KUKA KRL program: unicorn_3.src

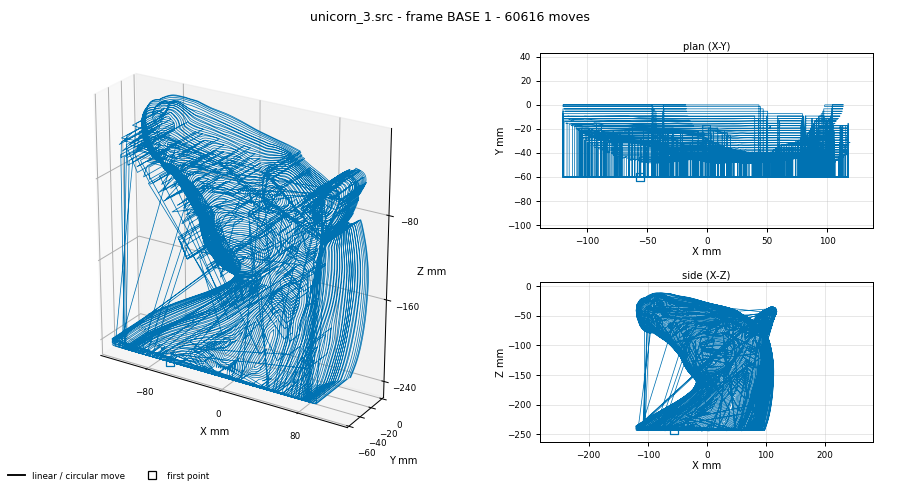
[picture p0: tool path of unicorn_3.src in frame BASE 1, 60616 of 60617 moves have a stored position in this frame; points joined in program order, loops and branches not executed]
&ACCESS RVP
&REL 1
&PARAM TEMPLATE = C:\KRC\Roboter\Template\vorgabe
&PARAM EDITMASK = *
DEF unicorn_3( )
EXT BAS (BAS_COMMAND :IN,REAL :IN )

INT INDX
FOR INDX=1 TO 6
	$ACC_AXIS[INDX]=50
	$VEL_AXIS[INDX]=20
ENDFOR

$VEL.ORI1=200
$VEL.ORI2=200
$ACC.ORI1=100
$ACC.ORI2=100

$VEL.CP = 0.2
$ACC.CP = 5

$IPO_MODE = #BASE
$APO.CDIS = 0.5
$ADVANCE = 5

$ACT_TOOL = 1
$TOOL=TOOL_DATA[1]
$ACT_BASE = 1
$BASE=BASE_DATA[1]

PTP {A1 30.0,A2 -100.0,A3 70.0,A4 0.0,A5 40.0,A6 0.0}

LIN {X -56.297,Y -60.000,Z -243.561,A -90.000,B 90.000,C 0.000} C_DIS
LIN {X -56.297,Y -47.308,Z -243.561,A -90.000,B 90.000,C 0.000} C_DIS
LIN {X -55.435,Y -47.308,Z -243.187,A -90.000,B 90.000,C 0.000} C_DIS
LIN {X -55.139,Y -47.308,Z -243.067,A -90.000,B 90.000,C 0.000} C_DIS
LIN {X -53.671,Y -47.308,Z -242.485,A -90.000,B 90.000,C 0.000} C_DIS
LIN {X -50.676,Y -47.308,Z -241.473,A -90.000,B 90.000,C 0.000} C_DIS
LIN {X -47.224,Y -47.308,Z -240.424,A -90.000,B 90.000,C 0.000} C_DIS
LIN {X -47.138,Y -47.308,Z -240.398,A -90.000,B 90.000,C 0.000} C_DIS
LIN {X -44.555,Y -47.308,Z -239.681,A -90.000,B 90.000,C 0.000} C_DIS
LIN {X -43.438,Y -47.308,Z -239.453,A -90.000,B 90.000,C 0.000} C_DIS
LIN {X -42.208,Y -47.308,Z -239.261,A -90.000,B 90.000,C 0.000} C_DIS
LIN {X -39.907,Y -47.308,Z -238.995,A -90.000,B 90.000,C 0.000} C_DIS
LIN {X -38.204,Y -47.308,Z -238.801,A -90.000,B 90.000,C 0.000} C_DIS
LIN {X -37.466,Y -47.308,Z -238.748,A -90.000,B 90.000,C 0.000} C_DIS
LIN {X -37.229,Y -47.308,Z -238.745,A -90.000,B 90.000,C 0.000} C_DIS
LIN {X -34.457,Y -47.308,Z -239.098,A -90.000,B 90.000,C 0.000} C_DIS
LIN {X -34.198,Y -47.308,Z -239.146,A -90.000,B 90.000,C 0.000} C_DIS
LIN {X -32.605,Y -47.308,Z -239.457,A -90.000,B 90.000,C 0.000} C_DIS
LIN {X -32.434,Y -47.308,Z -239.513,A -90.000,B 90.000,C 0.000} C_DIS
LIN {X -31.010,Y -47.308,Z -240.218,A -90.000,B 90.000,C 0.000} C_DIS
LIN {X -29.625,Y -47.308,Z -241.071,A -90.000,B 90.000,C 0.000} C_DIS
LIN {X -29.477,Y -47.308,Z -241.172,A -90.000,B 90.000,C 0.000} C_DIS
LIN {X -28.409,Y -47.308,Z -242.294,A -90.000,B 90.000,C 0.000} C_DIS
LIN {X -28.294,Y -47.308,Z -242.432,A -90.000,B 90.000,C 0.000} C_DIS
LIN {X -27.412,Y -47.308,Z -243.561,A -90.000,B 90.000,C 0.000} C_DIS
LIN {X -27.429,Y -47.311,Z -243.561,A -90.000,B 90.000,C 0.000} C_DIS
LIN {X -29.070,Y -47.511,Z -243.561,A -90.000,B 90.000,C 0.000} C_DIS
LIN {X -32.555,Y -47.888,Z -243.561,A -90.000,B 90.000,C 0.000} C_DIS
LIN {X -32.864,Y -47.915,Z -243.561,A -90.000,B 90.000,C 0.000} C_DIS
LIN {X -36.464,Y -48.174,Z -243.561,A -90.000,B 90.000,C 0.000} C_DIS
LIN {X -38.036,Y -48.261,Z -243.561,A -90.000,B 90.000,C 0.000} C_DIS
LIN {X -38.687,Y -48.281,Z -243.561,A -90.000,B 90.000,C 0.000} C_DIS
LIN {X -40.659,Y -48.330,Z -243.561,A -90.000,B 90.000,C 0.000} C_DIS
LIN {X -43.801,Y -48.366,Z -243.561,A -90.000,B 90.000,C 0.000} C_DIS
LIN {X -43.989,Y -48.366,Z -243.561,A -90.000,B 90.000,C 0.000} C_DIS
LIN {X -44.713,Y -48.344,Z -243.561,A -90.000,B 90.000,C 0.000} C_DIS
LIN {X -46.996,Y -48.250,Z -243.561,A -90.000,B 90.000,C 0.000} C_DIS
LIN {X -49.101,Y -48.148,Z -243.561,A -90.000,B 90.000,C 0.000} C_DIS
LIN {X -49.262,Y -48.138,Z -243.561,A -90.000,B 90.000,C 0.000} C_DIS
LIN {X -49.887,Y -48.091,Z -243.561,A -90.000,B 90.000,C 0.000} C_DIS
LIN {X -50.048,Y -48.076,Z -243.561,A -90.000,B 90.000,C 0.000} C_DIS
LIN {X -51.629,Y -47.893,Z -243.561,A -90.000,B 90.000,C 0.000} C_DIS
LIN {X -55.147,Y -47.500,Z -243.561,A -90.000,B 90.000,C 0.000} C_DIS
LIN {X -55.949,Y -47.375,Z -243.561,A -90.000,B 90.000,C 0.000} C_DIS
LIN {X -56.297,Y -47.308,Z -243.561,A -90.000,B 90.000,C 0.000} C_DIS
LIN {X -56.297,Y -60.000,Z -243.561,A -90.000,B 90.000,C 0.000} C_DIS
LIN {X -44.362,Y -60.000,Z -241.627,A -90.000,B 90.000,C 0.000} C_DIS
LIN {X -44.362,Y -47.846,Z -241.627,A -90.000,B 90.000,C 0.000} C_DIS
LIN {X -44.089,Y -47.838,Z -241.555,A -90.000,B 90.000,C 0.000} C_DIS
LIN {X -43.472,Y -47.831,Z -241.430,A -90.000,B 90.000,C 0.000} C_DIS
LIN {X -43.074,Y -47.823,Z -241.352,A -90.000,B 90.000,C 0.000} C_DIS
LIN {X -41.969,Y -47.812,Z -241.182,A -90.000,B 90.000,C 0.000} C_DIS
LIN {X -40.544,Y -47.812,Z -241.017,A -90.000,B 90.000,C 0.000} C_DIS
LIN {X -40.270,Y -47.806,Z -240.987,A -90.000,B 90.000,C 0.000} C_DIS
LIN {X -39.113,Y -47.767,Z -240.864,A -90.000,B 90.000,C 0.000} C_DIS
LIN {X -38.023,Y -47.717,Z -240.751,A -90.000,B 90.000,C 0.000} C_DIS
LIN {X -37.379,Y -47.693,Z -240.710,A -90.000,B 90.000,C 0.000} C_DIS
LIN {X -37.343,Y -47.692,Z -240.710,A -90.000,B 90.000,C 0.000} C_DIS
LIN {X -35.486,Y -47.692,Z -240.946,A -90.000,B 90.000,C 0.000} C_DIS
LIN {X -34.760,Y -47.683,Z -241.040,A -90.000,B 90.000,C 0.000} C_DIS
LIN {X -34.515,Y -47.679,Z -241.086,A -90.000,B 90.000,C 0.000} C_DIS
LIN {X -33.149,Y -47.622,Z -241.363,A -90.000,B 90.000,C 0.000} C_DIS
LIN {X -32.709,Y -47.622,Z -241.581,A -90.000,B 90.000,C 0.000} C_DIS
LIN {X -35.186,Y -47.796,Z -241.582,A -90.000,B 90.000,C 0.000} C_DIS
LIN {X -35.416,Y -47.809,Z -241.582,A -90.000,B 90.000,C 0.000} C_DIS
LIN {X -35.606,Y -47.816,Z -241.583,A -90.000,B 90.000,C 0.000} C_DIS
LIN {X -35.738,Y -47.821,Z -241.584,A -90.000,B 90.000,C 0.000} C_DIS
LIN {X -36.488,Y -47.842,Z -241.589,A -90.000,B 90.000,C 0.000} C_DIS
LIN {X -38.216,Y -47.887,Z -241.598,A -90.000,B 90.000,C 0.000} C_DIS
LIN {X -39.566,Y -47.921,Z -241.598,A -90.000,B 90.000,C 0.000} C_DIS
LIN {X -41.163,Y -47.939,Z -241.601,A -90.000,B 90.000,C 0.000} C_DIS
LIN {X -41.336,Y -47.939,Z -241.602,A -90.000,B 90.000,C 0.000} C_DIS
LIN {X -43.583,Y -47.877,Z -241.622,A -90.000,B 90.000,C 0.000} C_DIS
LIN {X -44.113,Y -47.856,Z -241.626,A -90.000,B 90.000,C 0.000} C_DIS
LIN {X -44.362,Y -47.846,Z -241.627,A -90.000,B 90.000,C 0.000} C_DIS
LIN {X -44.362,Y -60.000,Z -241.627,A -90.000,B 90.000,C 0.000} C_DIS
LIN {X 92.568,Y -60.000,Z -59.359,A -90.000,B 90.000,C 0.000} C_DIS
LIN {X 92.568,Y -51.610,Z -59.359,A -90.000,B 90.000,C 0.000} C_DIS
LIN {X 92.745,Y -51.646,Z -59.003,A -90.000,B 90.000,C 0.000} C_DIS
LIN {X 92.870,Y -51.669,Z -58.752,A -90.000,B 90.000,C 0.000} C_DIS
LIN {X 92.953,Y -51.684,Z -58.585,A -90.000,B 90.000,C 0.000} C_DIS
LIN {X 92.974,Y -51.688,Z -58.543,A -90.000,B 90.000,C 0.000} C_DIS
LIN {X 93.175,Y -51.715,Z -58.224,A -90.000,B 90.000,C 0.000} C_DIS
LIN {X 93.326,Y -51.727,Z -57.987,A -90.000,B 90.000,C 0.000} C_DIS
LIN {X 93.444,Y -51.726,Z -57.807,A -90.000,B 90.000,C 0.000} C_DIS
LIN {X 93.456,Y -51.725,Z -57.788,A -90.000,B 90.000,C 0.000} C_DIS
LIN {X 93.639,Y -51.720,Z -57.654,A -90.000,B 90.000,C 0.000} C_DIS
LIN {X 95.632,Y -51.629,Z -56.194,A -90.000,B 90.000,C 0.000} C_DIS
LIN {X 95.618,Y -51.636,Z -56.312,A -90.000,B 90.000,C 0.000} C_DIS
LIN {X 95.580,Y -51.642,Z -56.475,A -90.000,B 90.000,C 0.000} C_DIS
LIN {X 95.278,Y -51.660,Z -56.893,A -90.000,B 90.000,C 0.000} C_DIS
LIN {X 94.891,Y -51.678,Z -57.426,A -90.000,B 90.000,C 0.000} C_DIS
LIN {X 94.530,Y -51.696,Z -57.901,A -90.000,B 90.000,C 0.000} C_DIS
LIN {X 94.459,Y -51.699,Z -58.007,A -90.000,B 90.000,C 0.000} C_DIS
LIN {X 94.229,Y -51.708,Z -58.379,A -90.000,B 90.000,C 0.000} C_DIS
LIN {X 94.134,Y -51.708,Z -58.531,A -90.000,B 90.000,C 0.000} C_DIS
LIN {X 93.995,Y -51.711,Z -58.607,A -90.000,B 90.000,C 0.000} C_DIS
LIN {X 93.858,Y -51.710,Z -58.680,A -90.000,B 90.000,C 0.000} C_DIS
LIN {X 93.698,Y -51.705,Z -58.766,A -90.000,B 90.000,C 0.000} C_DIS
LIN {X 93.242,Y -51.670,Z -59.005,A -90.000,B 90.000,C 0.000} C_DIS
LIN {X 92.568,Y -51.610,Z -59.359,A -90.000,B 90.000,C 0.000} C_DIS
LIN {X 92.601,Y -51.623,Z -59.288,A -90.000,B 90.000,C 0.000} C_DIS
LIN {X 92.662,Y -51.637,Z -59.142,A -90.000,B 90.000,C 0.000} C_DIS
LIN {X 92.713,Y -51.650,Z -58.992,A -90.000,B 90.000,C 0.000} C_DIS
LIN {X 92.755,Y -51.661,Z -58.836,A -90.000,B 90.000,C 0.000} C_DIS
LIN {X 92.773,Y -51.666,Z -58.757,A -90.000,B 90.000,C 0.000} C_DIS
LIN {X 92.804,Y -51.673,Z -58.596,A -90.000,B 90.000,C 0.000} C_DIS
LIN {X 92.830,Y -51.679,Z -58.432,A -90.000,B 90.000,C 0.000} C_DIS
LIN {X 92.861,Y -51.683,Z -58.271,A -90.000,B 90.000,C 0.000} C_DIS
LIN {X 92.886,Y -51.683,Z -58.108,A -90.000,B 90.000,C 0.000} C_DIS
LIN {X 92.916,Y -51.679,Z -57.858,A -90.000,B 90.000,C 0.000} C_DIS
LIN {X 92.945,Y -51.662,Z -57.519,A -90.000,B 90.000,C 0.000} C_DIS
LIN {X 92.964,Y -51.658,Z -57.446,A -90.000,B 90.000,C 0.000} C_DIS
LIN {X 93.093,Y -51.597,Z -56.846,A -90.000,B 90.000,C 0.000} C_DIS
LIN {X 93.110,Y -51.588,Z -56.773,A -90.000,B 90.000,C 0.000} C_DIS
LIN {X 93.210,Y -51.543,Z -56.418,A -90.000,B 90.000,C 0.000} C_DIS
LIN {X 93.299,Y -51.507,Z -56.138,A -90.000,B 90.000,C 0.000} C_DIS
LIN {X 93.374,Y -51.480,Z -55.933,A -90.000,B 90.000,C 0.000} C_DIS
LIN {X 93.459,Y -51.453,Z -55.733,A -90.000,B 90.000,C 0.000} C_DIS
LIN {X 93.556,Y -51.427,Z -55.540,A -90.000,B 90.000,C 0.000} C_DIS
LIN {X 93.629,Y -51.409,Z -55.416,A -90.000,B 90.000,C 0.000} C_DIS
LIN {X 93.668,Y -51.400,Z -55.356,A -90.000,B 90.000,C 0.000} C_DIS
LIN {X 93.752,Y -51.382,Z -55.238,A -90.000,B 90.000,C 0.000} C_DIS
LIN {X 93.797,Y -51.373,Z -55.180,A -90.000,B 90.000,C 0.000} C_DIS
LIN {X 93.891,Y -51.356,Z -55.073,A -90.000,B 90.000,C 0.000} C_DIS
LIN {X 93.998,Y -51.337,Z -54.967,A -90.000,B 90.000,C 0.000} C_DIS
LIN {X 94.055,Y -51.328,Z -54.915,A -90.000,B 90.000,C 0.000} C_DIS
LIN {X 94.178,Y -51.308,Z -54.816,A -90.000,B 90.000,C 0.000} C_DIS
LIN {X 94.616,Y -51.308,Z -54.490,A -90.000,B 90.000,C 0.000} C_DIS
LIN {X 94.876,Y -51.308,Z -54.360,A -90.000,B 90.000,C 0.000} C_DIS
LIN {X 95.150,Y -51.308,Z -54.278,A -90.000,B 90.000,C 0.000} C_DIS
LIN {X 96.092,Y -51.308,Z -54.069,A -90.000,B 90.000,C 0.000} C_DIS
LIN {X 96.329,Y -51.308,Z -54.067,A -90.000,B 90.000,C 0.000} C_DIS
LIN {X 96.828,Y -51.308,Z -54.127,A -90.000,B 90.000,C 0.000} C_DIS
LIN {X 96.999,Y -51.308,Z -54.183,A -90.000,B 90.000,C 0.000} C_DIS
LIN {X 97.188,Y -51.308,Z -54.264,A -90.000,B 90.000,C 0.000} C_DIS
LIN {X 97.336,Y -51.308,Z -54.364,A -90.000,B 90.000,C 0.000} C_DIS
LIN {X 97.572,Y -51.308,Z -54.640,A -90.000,B 90.000,C 0.000} C_DIS
LIN {X 97.647,Y -51.308,Z -54.730,A -90.000,B 90.000,C 0.000} C_DIS
LIN {X 97.720,Y -51.308,Z -54.894,A -90.000,B 90.000,C 0.000} C_DIS
LIN {X 97.745,Y -51.308,Z -55.071,A -90.000,B 90.000,C 0.000} C_DIS
LIN {X 97.779,Y -51.308,Z -55.468,A -90.000,B 90.000,C 0.000} C_DIS
LIN {X 97.763,Y -51.308,Z -55.657,A -90.000,B 90.000,C 0.000} C_DIS
LIN {X 97.699,Y -51.308,Z -55.885,A -90.000,B 90.000,C 0.000} C_DIS
LIN {X 97.636,Y -51.308,Z -56.084,A -90.000,B 90.000,C 0.000} C_DIS
LIN {X 97.562,Y -51.308,Z -56.670,A -90.000,B 90.000,C 0.000} C_DIS
LIN {X 97.474,Y -51.308,Z -57.034,A -90.000,B 90.000,C 0.000} C_DIS
LIN {X 97.439,Y -51.308,Z -57.158,A -90.000,B 90.000,C 0.000} C_DIS
LIN {X 97.395,Y -51.308,Z -57.279,A -90.000,B 90.000,C 0.000} C_DIS
LIN {X 97.335,Y -51.308,Z -57.393,A -90.000,B 90.000,C 0.000} C_DIS
LIN {X 97.271,Y -51.308,Z -57.504,A -90.000,B 90.000,C 0.000} C_DIS
LIN {X 96.478,Y -51.308,Z -58.586,A -90.000,B 90.000,C 0.000} C_DIS
LIN {X 96.123,Y -51.308,Z -59.047,A -90.000,B 90.000,C 0.000} C_DIS
LIN {X 95.658,Y -51.308,Z -59.790,A -90.000,B 90.000,C 0.000} C_DIS
LIN {X 95.506,Y -51.308,Z -59.971,A -90.000,B 90.000,C 0.000} C_DIS
LIN {X 95.321,Y -51.308,Z -60.117,A -90.000,B 90.000,C 0.000} C_DIS
LIN {X 92.838,Y -51.308,Z -61.461,A -90.000,B 90.000,C 0.000} C_DIS
LIN {X 92.625,Y -51.308,Z -61.565,A -90.000,B 90.000,C 0.000} C_DIS
LIN {X 92.395,Y -51.308,Z -61.622,A -90.000,B 90.000,C 0.000} C_DIS
LIN {X 92.140,Y -51.308,Z -61.630,A -90.000,B 90.000,C 0.000} C_DIS
LIN {X 91.914,Y -51.308,Z -61.589,A -90.000,B 90.000,C 0.000} C_DIS
LIN {X 91.898,Y -51.308,Z -61.586,A -90.000,B 90.000,C 0.000} C_DIS
LIN {X 91.679,Y -51.308,Z -61.496,A -90.000,B 90.000,C 0.000} C_DIS
LIN {X 91.018,Y -51.308,Z -61.119,A -90.000,B 90.000,C 0.000} C_DIS
LIN {X 90.824,Y -51.308,Z -60.986,A -90.000,B 90.000,C 0.000} C_DIS
LIN {X 90.661,Y -51.308,Z -60.814,A -90.000,B 90.000,C 0.000} C_DIS
LIN {X 90.538,Y -51.308,Z -60.612,A -90.000,B 90.000,C 0.000} C_DIS
LIN {X 90.499,Y -51.308,Z -60.517,A -90.000,B 90.000,C 0.000} C_DIS
LIN {X 90.453,Y -51.308,Z -60.387,A -90.000,B 90.000,C 0.000} C_DIS
LIN {X 90.417,Y -51.308,Z -60.274,A -90.000,B 90.000,C 0.000} C_DIS
LIN {X 90.383,Y -51.308,Z -60.021,A -90.000,B 90.000,C 0.000} C_DIS
LIN {X 90.375,Y -51.308,Z -59.750,A -90.000,B 90.000,C 0.000} C_DIS
LIN {X 90.395,Y -51.308,Z -59.514,A -90.000,B 90.000,C 0.000} C_DIS
LIN {X 90.464,Y -51.308,Z -59.287,A -90.000,B 90.000,C 0.000} C_DIS
LIN {X 90.637,Y -51.308,Z -58.788,A -90.000,B 90.000,C 0.000} C_DIS
LIN {X 91.272,Y -51.308,Z -57.559,A -90.000,B 90.000,C 0.000} C_DIS
LIN {X 91.425,Y -51.308,Z -57.322,A -90.000,B 90.000,C 0.000} C_DIS
LIN {X 91.901,Y -51.308,Z -56.593,A -90.000,B 90.000,C 0.000} C_DIS
LIN {X 92.004,Y -51.308,Z -56.475,A -90.000,B 90.000,C 0.000} C_DIS
LIN {X 92.101,Y -51.308,Z -56.370,A -90.000,B 90.000,C 0.000} C_DIS
LIN {X 92.222,Y -51.308,Z -56.269,A -90.000,B 90.000,C 0.000} C_DIS
LIN {X 94.178,Y -51.308,Z -54.816,A -90.000,B 90.000,C 0.000} C_DIS
LIN {X 94.209,Y -51.312,Z -54.791,A -90.000,B 90.000,C 0.000} C_DIS
LIN {X 94.266,Y -51.308,Z -54.736,A -90.000,B 90.000,C 0.000} C_DIS
LIN {X 94.318,Y -51.301,Z -54.674,A -90.000,B 90.000,C 0.000} C_DIS
LIN {X 94.365,Y -51.290,Z -54.604,A -90.000,B 90.000,C 0.000} C_DIS
LIN {X 94.407,Y -51.276,Z -54.529,A -90.000,B 90.000,C 0.000} C_DIS
LIN {X 94.444,Y -51.260,Z -54.447,A -90.000,B 90.000,C 0.000} C_DIS
LIN {X 94.528,Y -51.204,Z -54.231,A -90.000,B 90.000,C 0.000} C_DIS
LIN {X 94.560,Y -51.177,Z -54.143,A -90.000,B 90.000,C 0.000} C_DIS
LIN {X 94.644,Y -51.086,Z -53.871,A -90.000,B 90.000,C 0.000} C_DIS
LIN {X 94.670,Y -51.055,Z -53.778,A -90.000,B 90.000,C 0.000} C_DIS
LIN {X 94.787,Y -50.899,Z -53.300,A -90.000,B 90.000,C 0.000} C_DIS
LIN {X 94.864,Y -50.807,Z -53.022,A -90.000,B 90.000,C 0.000} C_DIS
LIN {X 94.924,Y -50.748,Z -52.847,A -90.000,B 90.000,C 0.000} C_DIS
LIN {X 94.976,Y -50.707,Z -52.729,A -90.000,B 90.000,C 0.000} C_DIS
LIN {X 95.016,Y -50.681,Z -52.656,A -90.000,B 90.000,C 0.000} C_DIS
LIN {X 95.058,Y -50.656,Z -52.589,A -90.000,B 90.000,C 0.000} C_DIS
LIN {X 95.106,Y -50.631,Z -52.528,A -90.000,B 90.000,C 0.000} C_DIS
LIN {X 95.157,Y -50.607,Z -52.473,A -90.000,B 90.000,C 0.000} C_DIS
LIN {X 95.214,Y -50.584,Z -52.425,A -90.000,B 90.000,C 0.000} C_DIS
LIN {X 95.277,Y -50.560,Z -52.385,A -90.000,B 90.000,C 0.000} C_DIS
LIN {X 95.346,Y -50.536,Z -52.354,A -90.000,B 90.000,C 0.000} C_DIS
LIN {X 95.383,Y -50.524,Z -52.342,A -90.000,B 90.000,C 0.000} C_DIS
LIN {X 95.398,Y -50.526,Z -52.338,A -90.000,B 90.000,C 0.000} C_DIS
LIN {X 95.699,Y -50.560,Z -52.257,A -90.000,B 90.000,C 0.000} C_DIS
LIN {X 95.879,Y -50.584,Z -52.217,A -90.000,B 90.000,C 0.000} C_DIS
LIN {X 96.072,Y -50.619,Z -52.192,A -90.000,B 90.000,C 0.000} C_DIS
LIN {X 96.251,Y -50.654,Z -52.178,A -90.000,B 90.000,C 0.000} C_DIS
LIN {X 96.315,Y -50.664,Z -52.174,A -90.000,B 90.000,C 0.000} C_DIS
LIN {X 96.555,Y -50.706,Z -52.173,A -90.000,B 90.000,C 0.000} C_DIS
LIN {X 96.842,Y -50.762,Z -52.191,A -90.000,B 90.000,C 0.000} C_DIS
LIN {X 96.936,Y -50.779,Z -52.197,A -90.000,B 90.000,C 0.000} C_DIS
LIN {X 97.072,Y -50.798,Z -52.208,A -90.000,B 90.000,C 0.000} C_DIS
LIN {X 97.235,Y -50.822,Z -52.230,A -90.000,B 90.000,C 0.000} C_DIS
LIN {X 97.288,Y -50.829,Z -52.240,A -90.000,B 90.000,C 0.000} C_DIS
LIN {X 97.451,Y -50.854,Z -52.281,A -90.000,B 90.000,C 0.000} C_DIS
LIN {X 97.636,Y -50.884,Z -52.335,A -90.000,B 90.000,C 0.000} C_DIS
LIN {X 97.768,Y -50.897,Z -52.383,A -90.000,B 90.000,C 0.000} C_DIS
LIN {X 97.864,Y -50.907,Z -52.422,A -90.000,B 90.000,C 0.000} C_DIS
LIN {X 97.959,Y -50.913,Z -52.461,A -90.000,B 90.000,C 0.000} C_DIS
LIN {X 98.051,Y -50.919,Z -52.502,A -90.000,B 90.000,C 0.000} C_DIS
LIN {X 98.097,Y -50.923,Z -52.524,A -90.000,B 90.000,C 0.000} C_DIS
LIN {X 98.193,Y -50.933,Z -52.576,A -90.000,B 90.000,C 0.000} C_DIS
LIN {X 98.271,Y -50.942,Z -52.623,A -90.000,B 90.000,C 0.000} C_DIS
LIN {X 98.456,Y -50.952,Z -52.746,A -90.000,B 90.000,C 0.000} C_DIS
LIN {X 98.501,Y -50.952,Z -52.778,A -90.000,B 90.000,C 0.000} C_DIS
LIN {X 98.610,Y -50.953,Z -52.864,A -90.000,B 90.000,C 0.000} C_DIS
LIN {X 98.641,Y -50.954,Z -52.891,A -90.000,B 90.000,C 0.000} C_DIS
LIN {X 98.705,Y -50.952,Z -52.950,A -90.000,B 90.000,C 0.000} C_DIS
LIN {X 98.809,Y -50.952,Z -53.059,A -90.000,B 90.000,C 0.000} C_DIS
LIN {X 99.055,Y -50.948,Z -53.347,A -90.000,B 90.000,C 0.000} C_DIS
LIN {X 99.196,Y -50.939,Z -53.520,A -90.000,B 90.000,C 0.000} C_DIS
LIN {X 99.250,Y -50.934,Z -53.594,A -90.000,B 90.000,C 0.000} C_DIS
LIN {X 99.296,Y -50.928,Z -53.664,A -90.000,B 90.000,C 0.000} C_DIS
LIN {X 99.365,Y -50.920,Z -53.781,A -90.000,B 90.000,C 0.000} C_DIS
LIN {X 99.410,Y -50.911,Z -53.872,A -90.000,B 90.000,C 0.000} C_DIS
LIN {X 99.508,Y -50.891,Z -54.101,A -90.000,B 90.000,C 0.000} C_DIS
LIN {X 99.574,Y -50.876,Z -54.280,A -90.000,B 90.000,C 0.000} C_DIS
LIN {X 99.601,Y -50.865,Z -54.378,A -90.000,B 90.000,C 0.000} C_DIS
LIN {X 99.621,Y -50.850,Z -54.474,A -90.000,B 90.000,C 0.000} C_DIS
LIN {X 99.639,Y -50.841,Z -54.578,A -90.000,B 90.000,C 0.000} C_DIS
LIN {X 99.671,Y -50.821,Z -54.837,A -90.000,B 90.000,C 0.000} C_DIS
LIN {X 99.683,Y -50.811,Z -54.996,A -90.000,B 90.000,C 0.000} C_DIS
LIN {X 99.703,Y -50.785,Z -55.307,A -90.000,B 90.000,C 0.000} C_DIS
LIN {X 99.697,Y -50.751,Z -55.568,A -90.000,B 90.000,C 0.000} C_DIS
LIN {X 99.668,Y -50.720,Z -55.818,A -90.000,B 90.000,C 0.000} C_DIS
LIN {X 99.647,Y -50.705,Z -55.953,A -90.000,B 90.000,C 0.000} C_DIS
LIN {X 99.614,Y -50.692,Z -56.100,A -90.000,B 90.000,C 0.000} C_DIS
LIN {X 99.527,Y -50.673,Z -56.389,A -90.000,B 90.000,C 0.000} C_DIS
LIN {X 99.494,Y -50.667,Z -56.491,A -90.000,B 90.000,C 0.000} C_DIS
LIN {X 99.480,Y -50.658,Z -56.578,A -90.000,B 90.000,C 0.000} C_DIS
LIN {X 99.413,Y -50.624,Z -56.993,A -90.000,B 90.000,C 0.000} C_DIS
LIN {X 99.380,Y -50.616,Z -57.135,A -90.000,B 90.000,C 0.000} C_DIS
LIN {X 99.310,Y -50.598,Z -57.393,A -90.000,B 90.000,C 0.000} C_DIS
LIN {X 99.255,Y -50.580,Z -57.579,A -90.000,B 90.000,C 0.000} C_DIS
LIN {X 99.220,Y -50.571,Z -57.689,A -90.000,B 90.000,C 0.000} C_DIS
LIN {X 99.158,Y -50.567,Z -57.865,A -90.000,B 90.000,C 0.000} C_DIS
LIN {X 99.137,Y -50.567,Z -57.923,A -90.000,B 90.000,C 0.000} C_DIS
LIN {X 99.056,Y -50.570,Z -58.113,A -90.000,B 90.000,C 0.000} C_DIS
LIN {X 98.948,Y -50.580,Z -58.324,A -90.000,B 90.000,C 0.000} C_DIS
LIN {X 98.834,Y -50.590,Z -58.524,A -90.000,B 90.000,C 0.000} C_DIS
LIN {X 98.810,Y -50.593,Z -58.562,A -90.000,B 90.000,C 0.000} C_DIS
LIN {X 98.626,Y -50.600,Z -58.820,A -90.000,B 90.000,C 0.000} C_DIS
LIN {X 98.455,Y -50.599,Z -59.052,A -90.000,B 90.000,C 0.000} C_DIS
LIN {X 97.963,Y -50.613,Z -59.733,A -90.000,B 90.000,C 0.000} C_DIS
LIN {X 97.668,Y -50.626,Z -60.122,A -90.000,B 90.000,C 0.000} C_DIS
LIN {X 97.412,Y -50.622,Z -60.527,A -90.000,B 90.000,C 0.000} C_DIS
LIN {X 97.250,Y -50.616,Z -60.784,A -90.000,B 90.000,C 0.000} C_DIS
LIN {X 97.107,Y -50.621,Z -60.985,A -90.000,B 90.000,C 0.000} C_DIS
LIN {X 97.084,Y -50.622,Z -61.013,A -90.000,B 90.000,C 0.000} C_DIS
LIN {X 96.902,Y -50.619,Z -61.228,A -90.000,B 90.000,C 0.000} C_DIS
LIN {X 96.862,Y -50.619,Z -61.270,A -90.000,B 90.000,C 0.000} C_DIS
LIN {X 96.805,Y -50.616,Z -61.326,A -90.000,B 90.000,C 0.000} C_DIS
LIN {X 96.663,Y -50.615,Z -61.448,A -90.000,B 90.000,C 0.000} C_DIS
LIN {X 96.417,Y -50.620,Z -61.641,A -90.000,B 90.000,C 0.000} C_DIS
LIN {X 96.326,Y -50.624,Z -61.705,A -90.000,B 90.000,C 0.000} C_DIS
LIN {X 96.217,Y -50.632,Z -61.772,A -90.000,B 90.000,C 0.000} C_DIS
LIN {X 94.915,Y -50.736,Z -62.516,A -90.000,B 90.000,C 0.000} C_DIS
LIN {X 94.357,Y -50.764,Z -62.827,A -90.000,B 90.000,C 0.000} C_DIS
LIN {X 94.108,Y -50.765,Z -62.962,A -90.000,B 90.000,C 0.000} C_DIS
LIN {X 93.876,Y -50.752,Z -63.083,A -90.000,B 90.000,C 0.000} C_DIS
LIN {X 93.676,Y -50.727,Z -63.181,A -90.000,B 90.000,C 0.000} C_DIS
LIN {X 93.468,Y -50.706,Z -63.275,A -90.000,B 90.000,C 0.000} C_DIS
LIN {X 93.374,Y -50.697,Z -63.315,A -90.000,B 90.000,C 0.000} C_DIS
LIN {X 93.320,Y -50.692,Z -63.336,A -90.000,B 90.000,C 0.000} C_DIS
LIN {X 93.081,Y -50.681,Z -63.408,A -90.000,B 90.000,C 0.000} C_DIS
LIN {X 92.834,Y -50.676,Z -63.467,A -90.000,B 90.000,C 0.000} C_DIS
LIN {X 92.710,Y -50.675,Z -63.492,A -90.000,B 90.000,C 0.000} C_DIS
LIN {X 92.439,Y -50.684,Z -63.521,A -90.000,B 90.000,C 0.000} C_DIS
LIN {X 92.191,Y -50.695,Z -63.533,A -90.000,B 90.000,C 0.000} C_DIS
LIN {X 92.043,Y -50.695,Z -63.531,A -90.000,B 90.000,C 0.000} C_DIS
LIN {X 91.915,Y -50.697,Z -63.521,A -90.000,B 90.000,C 0.000} C_DIS
LIN {X 91.790,Y -50.698,Z -63.502,A -90.000,B 90.000,C 0.000} C_DIS
LIN {X 91.504,Y -50.701,Z -63.450,A -90.000,B 90.000,C 0.000} C_DIS
LIN {X 91.501,Y -50.701,Z -63.450,A -90.000,B 90.000,C 0.000} C_DIS
LIN {X 91.290,Y -50.709,Z -63.394,A -90.000,B 90.000,C 0.000} C_DIS
LIN {X 91.171,Y -50.721,Z -63.354,A -90.000,B 90.000,C 0.000} C_DIS
LIN {X 90.938,Y -50.748,Z -63.267,A -90.000,B 90.000,C 0.000} C_DIS
LIN {X 90.853,Y -50.753,Z -63.231,A -90.000,B 90.000,C 0.000} C_DIS
LIN {X 90.710,Y -50.766,Z -63.160,A -90.000,B 90.000,C 0.000} C_DIS
LIN {X 90.514,Y -50.783,Z -63.053,A -90.000,B 90.000,C 0.000} C_DIS
LIN {X 90.315,Y -50.791,Z -62.942,A -90.000,B 90.000,C 0.000} C_DIS
LIN {X 90.061,Y -50.784,Z -62.795,A -90.000,B 90.000,C 0.000} C_DIS
LIN {X 89.938,Y -50.780,Z -62.717,A -90.000,B 90.000,C 0.000} C_DIS
LIN {X 89.675,Y -50.776,Z -62.534,A -90.000,B 90.000,C 0.000} C_DIS
LIN {X 89.573,Y -50.779,Z -62.454,A -90.000,B 90.000,C 0.000} C_DIS
LIN {X 89.481,Y -50.783,Z -62.371,A -90.000,B 90.000,C 0.000} C_DIS
LIN {X 89.316,Y -50.783,Z -62.200,A -90.000,B 90.000,C 0.000} C_DIS
LIN {X 89.203,Y -50.774,Z -62.074,A -90.000,B 90.000,C 0.000} C_DIS
LIN {X 89.142,Y -50.769,Z -61.997,A -90.000,B 90.000,C 0.000} C_DIS
LIN {X 89.101,Y -50.764,Z -61.941,A -90.000,B 90.000,C 0.000} C_DIS
LIN {X 89.021,Y -50.755,Z -61.816,A -90.000,B 90.000,C 0.000} C_DIS
LIN {X 88.901,Y -50.739,Z -61.611,A -90.000,B 90.000,C 0.000} C_DIS
LIN {X 88.873,Y -50.732,Z -61.559,A -90.000,B 90.000,C 0.000} C_DIS
LIN {X 88.830,Y -50.721,Z -61.472,A -90.000,B 90.000,C 0.000} C_DIS
LIN {X 88.800,Y -50.714,Z -61.405,A -90.000,B 90.000,C 0.000} C_DIS
LIN {X 88.737,Y -50.700,Z -61.242,A -90.000,B 90.000,C 0.000} C_DIS
LIN {X 88.704,Y -50.690,Z -61.146,A -90.000,B 90.000,C 0.000} C_DIS
LIN {X 88.616,Y -50.664,Z -60.859,A -90.000,B 90.000,C 0.000} C_DIS
LIN {X 88.597,Y -50.659,Z -60.790,A -90.000,B 90.000,C 0.000} C_DIS
LIN {X 88.571,Y -50.648,Z -60.673,A -90.000,B 90.000,C 0.000} C_DIS
LIN {X 88.557,Y -50.641,Z -60.582,A -90.000,B 90.000,C 0.000} C_DIS
LIN {X 88.523,Y -50.625,Z -60.292,A -90.000,B 90.000,C 0.000} C_DIS
LIN {X 88.512,Y -50.614,Z -60.152,A -90.000,B 90.000,C 0.000} C_DIS
LIN {X 88.509,Y -50.608,Z -60.025,A -90.000,B 90.000,C 0.000} C_DIS
LIN {X 88.513,Y -50.581,Z -59.797,A -90.000,B 90.000,C 0.000} C_DIS
LIN {X 88.517,Y -50.571,Z -59.696,A -90.000,B 90.000,C 0.000} C_DIS
LIN {X 88.526,Y -50.563,Z -59.594,A -90.000,B 90.000,C 0.000} C_DIS
LIN {X 88.552,Y -50.548,Z -59.358,A -90.000,B 90.000,C 0.000} C_DIS
LIN {X 88.571,Y -50.542,Z -59.223,A -90.000,B 90.000,C 0.000} C_DIS
LIN {X 88.584,Y -50.536,Z -59.162,A -90.000,B 90.000,C 0.000} C_DIS
LIN {X 88.634,Y -50.526,Z -58.979,A -90.000,B 90.000,C 0.000} C_DIS
LIN {X 88.728,Y -50.519,Z -58.686,A -90.000,B 90.000,C 0.000} C_DIS
LIN {X 88.799,Y -50.516,Z -58.484,A -90.000,B 90.000,C 0.000} C_DIS
LIN {X 88.895,Y -50.501,Z -58.229,A -90.000,B 90.000,C 0.000} C_DIS
LIN {X 88.940,Y -50.490,Z -58.119,A -90.000,B 90.000,C 0.000} C_DIS
LIN {X 89.022,Y -50.476,Z -57.953,A -90.000,B 90.000,C 0.000} C_DIS
LIN {X 89.073,Y -50.470,Z -57.861,A -90.000,B 90.000,C 0.000} C_DIS
LIN {X 89.242,Y -50.440,Z -57.563,A -90.000,B 90.000,C 0.000} C_DIS
LIN {X 89.712,Y -50.351,Z -56.753,A -90.000,B 90.000,C 0.000} C_DIS
LIN {X 89.781,Y -50.341,Z -56.642,A -90.000,B 90.000,C 0.000} C_DIS
LIN {X 89.964,Y -50.318,Z -56.381,A -90.000,B 90.000,C 0.000} C_DIS
LIN {X 90.495,Y -50.257,Z -55.634,A -90.000,B 90.000,C 0.000} C_DIS
LIN {X 90.594,Y -50.253,Z -55.508,A -90.000,B 90.000,C 0.000} C_DIS
LIN {X 90.759,Y -50.254,Z -55.317,A -90.000,B 90.000,C 0.000} C_DIS
LIN {X 90.915,Y -50.259,Z -55.148,A -90.000,B 90.000,C 0.000} C_DIS
LIN {X 91.008,Y -50.259,Z -55.065,A -90.000,B 90.000,C 0.000} C_DIS
LIN {X 91.127,Y -50.261,Z -54.963,A -90.000,B 90.000,C 0.000} C_DIS
LIN {X 91.217,Y -50.265,Z -54.890,A -90.000,B 90.000,C 0.000} C_DIS
LIN {X 93.428,Y -50.338,Z -53.194,A -90.000,B 90.000,C 0.000} C_DIS
LIN {X 93.631,Y -50.333,Z -53.048,A -90.000,B 90.000,C 0.000} C_DIS
LIN {X 93.746,Y -50.337,Z -52.974,A -90.000,B 90.000,C 0.000} C_DIS
LIN {X 93.834,Y -50.340,Z -52.925,A -90.000,B 90.000,C 0.000} C_DIS
LIN {X 94.152,Y -50.359,Z -52.756,A -90.000,B 90.000,C 0.000} C_DIS
LIN {X 94.241,Y -50.368,Z -52.713,A -90.000,B 90.000,C 0.000} C_DIS
LIN {X 94.368,Y -50.380,Z -52.663,A -90.000,B 90.000,C 0.000} C_DIS
LIN {X 94.701,Y -50.420,Z -52.543,A -90.000,B 90.000,C 0.000} C_DIS
LIN {X 95.227,Y -50.502,Z -52.386,A -90.000,B 90.000,C 0.000} C_DIS
LIN {X 95.383,Y -50.524,Z -52.342,A -90.000,B 90.000,C 0.000} C_DIS
LIN {X 95.355,Y -50.381,Z -52.093,A -90.000,B 90.000,C 0.000} C_DIS
LIN {X 95.340,Y -50.220,Z -51.838,A -90.000,B 90.000,C 0.000} C_DIS
LIN {X 95.324,Y -50.015,Z -51.544,A -90.000,B 90.000,C 0.000} C_DIS
LIN {X 95.307,Y -49.784,Z -51.251,A -90.000,B 90.000,C 0.000} C_DIS
LIN {X 95.293,Y -49.558,Z -50.995,A -90.000,B 90.000,C 0.000} C_DIS
LIN {X 95.293,Y -49.308,Z -50.744,A -90.000,B 90.000,C 0.000} C_DIS
LIN {X 95.463,Y -49.358,Z -50.676,A -90.000,B 90.000,C 0.000} C_DIS
LIN {X 95.589,Y -49.395,Z -50.632,A -90.000,B 90.000,C 0.000} C_DIS
LIN {X 95.751,Y -49.434,Z -50.586,A -90.000,B 90.000,C 0.000} C_DIS
LIN {X 95.863,Y -49.466,Z -50.559,A -90.000,B 90.000,C 0.000} C_DIS
LIN {X 96.059,Y -49.526,Z -50.517,A -90.000,B 90.000,C 0.000} C_DIS
LIN {X 96.135,Y -49.551,Z -50.502,A -90.000,B 90.000,C 0.000} C_DIS
LIN {X 96.294,Y -49.606,Z -50.475,A -90.000,B 90.000,C 0.000} C_DIS
LIN {X 96.463,Y -49.658,Z -50.451,A -90.000,B 90.000,C 0.000} C_DIS
LIN {X 96.690,Y -49.729,Z -50.434,A -90.000,B 90.000,C 0.000} C_DIS
LIN {X 96.856,Y -49.783,Z -50.425,A -90.000,B 90.000,C 0.000} C_DIS
LIN {X 97.045,Y -49.849,Z -50.421,A -90.000,B 90.000,C 0.000} C_DIS
LIN {X 97.319,Y -49.923,Z -50.427,A -90.000,B 90.000,C 0.000} C_DIS
LIN {X 97.431,Y -49.954,Z -50.431,A -90.000,B 90.000,C 0.000} C_DIS
LIN {X 97.593,Y -50.002,Z -50.441,A -90.000,B 90.000,C 0.000} C_DIS
LIN {X 97.723,Y -50.037,Z -50.456,A -90.000,B 90.000,C 0.000} C_DIS
LIN {X 97.760,Y -50.048,Z -50.460,A -90.000,B 90.000,C 0.000} C_DIS
LIN {X 97.935,Y -50.093,Z -50.494,A -90.000,B 90.000,C 0.000} C_DIS
LIN {X 98.106,Y -50.139,Z -50.532,A -90.000,B 90.000,C 0.000} C_DIS
LIN {X 98.202,Y -50.166,Z -50.555,A -90.000,B 90.000,C 0.000} C_DIS
LIN {X 98.376,Y -50.207,Z -50.604,A -90.000,B 90.000,C 0.000} C_DIS
LIN {X 98.486,Y -50.234,Z -50.638,A -90.000,B 90.000,C 0.000} C_DIS
LIN {X 98.772,Y -50.293,Z -50.743,A -90.000,B 90.000,C 0.000} C_DIS
LIN {X 98.974,Y -50.336,Z -50.826,A -90.000,B 90.000,C 0.000} C_DIS
LIN {X 99.109,Y -50.369,Z -50.890,A -90.000,B 90.000,C 0.000} C_DIS
LIN {X 99.198,Y -50.391,Z -50.934,A -90.000,B 90.000,C 0.000} C_DIS
LIN {X 99.380,Y -50.422,Z -51.042,A -90.000,B 90.000,C 0.000} C_DIS
LIN {X 99.626,Y -50.455,Z -51.201,A -90.000,B 90.000,C 0.000} C_DIS
LIN {X 99.761,Y -50.474,Z -51.298,A -90.000,B 90.000,C 0.000} C_DIS
LIN {X 99.936,Y -50.489,Z -51.439,A -90.000,B 90.000,C 0.000} C_DIS
LIN {X 100.050,Y -50.493,Z -51.544,A -90.000,B 90.000,C 0.000} C_DIS
LIN {X 100.107,Y -50.495,Z -51.600,A -90.000,B 90.000,C 0.000} C_DIS
LIN {X 100.258,Y -50.494,Z -51.759,A -90.000,B 90.000,C 0.000} C_DIS
LIN {X 100.425,Y -50.484,Z -51.956,A -90.000,B 90.000,C 0.000} C_DIS
LIN {X 100.587,Y -50.464,Z -52.154,A -90.000,B 90.000,C 0.000} C_DIS
LIN {X 100.684,Y -50.453,Z -52.275,A -90.000,B 90.000,C 0.000} C_DIS
LIN {X 100.809,Y -50.435,Z -52.445,A -90.000,B 90.000,C 0.000} C_DIS
LIN {X 100.911,Y -50.412,Z -52.603,A -90.000,B 90.000,C 0.000} C_DIS
LIN {X 100.999,Y -50.391,Z -52.756,A -90.000,B 90.000,C 0.000} C_DIS
LIN {X 101.066,Y -50.374,Z -52.882,A -90.000,B 90.000,C 0.000} C_DIS
LIN {X 101.118,Y -50.354,Z -52.994,A -90.000,B 90.000,C 0.000} C_DIS
LIN {X 101.193,Y -50.311,Z -53.183,A -90.000,B 90.000,C 0.000} C_DIS
LIN {X 101.253,Y -50.275,Z -53.343,A -90.000,B 90.000,C 0.000} C_DIS
LIN {X 101.301,Y -50.244,Z -53.488,A -90.000,B 90.000,C 0.000} C_DIS
LIN {X 101.335,Y -50.219,Z -53.598,A -90.000,B 90.000,C 0.000} C_DIS
LIN {X 101.366,Y -50.197,Z -53.709,A -90.000,B 90.000,C 0.000} C_DIS
LIN {X 101.411,Y -50.168,Z -53.890,A -90.000,B 90.000,C 0.000} C_DIS
LIN {X 101.440,Y -50.149,Z -54.029,A -90.000,B 90.000,C 0.000} C_DIS
LIN {X 101.468,Y -50.110,Z -54.231,A -90.000,B 90.000,C 0.000} C_DIS
LIN {X 101.491,Y -50.048,Z -54.538,A -90.000,B 90.000,C 0.000} C_DIS
LIN {X 101.498,Y -50.019,Z -54.693,A -90.000,B 90.000,C 0.000} C_DIS
LIN {X 101.501,Y -50.000,Z -54.800,A -90.000,B 90.000,C 0.000} C_DIS
LIN {X 101.511,Y -49.950,Z -55.122,A -90.000,B 90.000,C 0.000} C_DIS
LIN {X 101.511,Y -49.934,Z -55.236,A -90.000,B 90.000,C 0.000} C_DIS
LIN {X 101.504,Y -49.892,Z -55.556,A -90.000,B 90.000,C 0.000} C_DIS
LIN {X 101.492,Y -49.874,Z -55.671,A -90.000,B 90.000,C 0.000} C_DIS
LIN {X 101.478,Y -49.858,Z -55.785,A -90.000,B 90.000,C 0.000} C_DIS
LIN {X 101.458,Y -49.841,Z -55.965,A -90.000,B 90.000,C 0.000} C_DIS
LIN {X 101.433,Y -49.826,Z -56.148,A -90.000,B 90.000,C 0.000} C_DIS
LIN {X 101.380,Y -49.813,Z -56.424,A -90.000,B 90.000,C 0.000} C_DIS
LIN {X 101.342,Y -49.809,Z -56.582,A -90.000,B 90.000,C 0.000} C_DIS
LIN {X 101.265,Y -49.795,Z -56.843,A -90.000,B 90.000,C 0.000} C_DIS
LIN {X 101.244,Y -49.781,Z -56.965,A -90.000,B 90.000,C 0.000} C_DIS
LIN {X 101.196,Y -49.745,Z -57.209,A -90.000,B 90.000,C 0.000} C_DIS
LIN {X 101.179,Y -49.733,Z -57.291,A -90.000,B 90.000,C 0.000} C_DIS
LIN {X 101.114,Y -49.705,Z -57.538,A -90.000,B 90.000,C 0.000} C_DIS
LIN {X 101.055,Y -49.686,Z -57.748,A -90.000,B 90.000,C 0.000} C_DIS
LIN {X 100.971,Y -49.665,Z -58.047,A -90.000,B 90.000,C 0.000} C_DIS
LIN {X 100.938,Y -49.659,Z -58.158,A -90.000,B 90.000,C 0.000} C_DIS
LIN {X 100.903,Y -49.654,Z -58.262,A -90.000,B 90.000,C 0.000} C_DIS
LIN {X 100.808,Y -49.647,Z -58.525,A -90.000,B 90.000,C 0.000} C_DIS
LIN {X 100.765,Y -49.646,Z -58.633,A -90.000,B 90.000,C 0.000} C_DIS
LIN {X 100.682,Y -49.648,Z -58.823,A -90.000,B 90.000,C 0.000} C_DIS
LIN {X 100.619,Y -49.651,Z -58.957,A -90.000,B 90.000,C 0.000} C_DIS
LIN {X 100.511,Y -49.661,Z -59.168,A -90.000,B 90.000,C 0.000} C_DIS
LIN {X 100.387,Y -49.676,Z -59.393,A -90.000,B 90.000,C 0.000} C_DIS
LIN {X 100.306,Y -49.687,Z -59.532,A -90.000,B 90.000,C 0.000} C_DIS
LIN {X 100.226,Y -49.698,Z -59.656,A -90.000,B 90.000,C 0.000} C_DIS
LIN {X 99.416,Y -49.753,Z -60.803,A -90.000,B 90.000,C 0.000} C_DIS
LIN {X 99.154,Y -49.775,Z -61.159,A -90.000,B 90.000,C 0.000} C_DIS
LIN {X 98.773,Y -49.781,Z -61.774,A -90.000,B 90.000,C 0.000} C_DIS
LIN {X 98.651,Y -49.785,Z -61.950,A -90.000,B 90.000,C 0.000} C_DIS
LIN {X 98.588,Y -49.787,Z -62.040,A -90.000,B 90.000,C 0.000} C_DIS
LIN {X 98.543,Y -49.785,Z -62.099,A -90.000,B 90.000,C 0.000} C_DIS
LIN {X 98.325,Y -49.784,Z -62.358,A -90.000,B 90.000,C 0.000} C_DIS
LIN {X 98.199,Y -49.783,Z -62.501,A -90.000,B 90.000,C 0.000} C_DIS
LIN {X 98.052,Y -49.786,Z -62.651,A -90.000,B 90.000,C 0.000} C_DIS
LIN {X 97.865,Y -49.795,Z -62.820,A -90.000,B 90.000,C 0.000} C_DIS
LIN {X 97.780,Y -49.800,Z -62.894,A -90.000,B 90.000,C 0.000} C_DIS
LIN {X 97.500,Y -49.822,Z -63.122,A -90.000,B 90.000,C 0.000} C_DIS
LIN {X 97.385,Y -49.835,Z -63.207,A -90.000,B 90.000,C 0.000} C_DIS
LIN {X 97.253,Y -49.851,Z -63.299,A -90.000,B 90.000,C 0.000} C_DIS
LIN {X 97.099,Y -49.872,Z -63.398,A -90.000,B 90.000,C 0.000} C_DIS
LIN {X 96.926,Y -49.899,Z -63.503,A -90.000,B 90.000,C 0.000} C_DIS
LIN {X 96.204,Y -49.976,Z -63.924,A -90.000,B 90.000,C 0.000} C_DIS
LIN {X 95.906,Y -50.001,Z -64.095,A -90.000,B 90.000,C 0.000} C_DIS
LIN {X 95.621,Y -50.005,Z -64.250,A -90.000,B 90.000,C 0.000} C_DIS
LIN {X 95.218,Y -50.009,Z -64.466,A -90.000,B 90.000,C 0.000} C_DIS
LIN {X 94.580,Y -49.976,Z -64.799,A -90.000,B 90.000,C 0.000} C_DIS
LIN {X 94.503,Y -49.973,Z -64.839,A -90.000,B 90.000,C 0.000} C_DIS
LIN {X 94.193,Y -49.961,Z -64.985,A -90.000,B 90.000,C 0.000} C_DIS
LIN {X 94.062,Y -49.959,Z -65.042,A -90.000,B 90.000,C 0.000} C_DIS
LIN {X 93.971,Y -49.958,Z -65.078,A -90.000,B 90.000,C 0.000} C_DIS
LIN {X 93.900,Y -49.958,Z -65.104,A -90.000,B 90.000,C 0.000} C_DIS
LIN {X 93.649,Y -49.959,Z -65.185,A -90.000,B 90.000,C 0.000} C_DIS
LIN {X 93.537,Y -49.960,Z -65.217,A -90.000,B 90.000,C 0.000} C_DIS
LIN {X 93.207,Y -49.966,Z -65.300,A -90.000,B 90.000,C 0.000} C_DIS
LIN {X 93.082,Y -49.970,Z -65.327,A -90.000,B 90.000,C 0.000} C_DIS
LIN {X 92.887,Y -49.980,Z -65.359,A -90.000,B 90.000,C 0.000} C_DIS
LIN {X 92.823,Y -49.984,Z -65.367,A -90.000,B 90.000,C 0.000} C_DIS
LIN {X 92.542,Y -49.993,Z -65.395,A -90.000,B 90.000,C 0.000} C_DIS
LIN {X 92.238,Y -50.008,Z -65.411,A -90.000,B 90.000,C 0.000} C_DIS
LIN {X 92.020,Y -50.013,Z -65.411,A -90.000,B 90.000,C 0.000} C_DIS
LIN {X 91.882,Y -50.014,Z -65.405,A -90.000,B 90.000,C 0.000} C_DIS
LIN {X 91.733,Y -50.017,Z -65.393,A -90.000,B 90.000,C 0.000} C_DIS
LIN {X 91.555,Y -50.019,Z -65.370,A -90.000,B 90.000,C 0.000} C_DIS
LIN {X 91.390,Y -50.024,Z -65.343,A -90.000,B 90.000,C 0.000} C_DIS
LIN {X 91.096,Y -50.033,Z -65.291,A -90.000,B 90.000,C 0.000} C_DIS
LIN {X 90.964,Y -50.041,Z -65.260,A -90.000,B 90.000,C 0.000} C_DIS
LIN {X 90.790,Y -50.052,Z -65.216,A -90.000,B 90.000,C 0.000} C_DIS
LIN {X 90.645,Y -50.064,Z -65.174,A -90.000,B 90.000,C 0.000} C_DIS
LIN {X 90.443,Y -50.072,Z -65.100,A -90.000,B 90.000,C 0.000} C_DIS
LIN {X 90.358,Y -50.077,Z -65.067,A -90.000,B 90.000,C 0.000} C_DIS
LIN {X 90.281,Y -50.079,Z -65.035,A -90.000,B 90.000,C 0.000} C_DIS
LIN {X 90.093,Y -50.082,Z -64.954,A -90.000,B 90.000,C 0.000} C_DIS
LIN {X 90.015,Y -50.083,Z -64.918,A -90.000,B 90.000,C 0.000} C_DIS
LIN {X 89.767,Y -50.100,Z -64.792,A -90.000,B 90.000,C 0.000} C_DIS
LIN {X 89.503,Y -50.122,Z -64.649,A -90.000,B 90.000,C 0.000} C_DIS
LIN {X 89.230,Y -50.135,Z -64.498,A -90.000,B 90.000,C 0.000} C_DIS
LIN {X 89.066,Y -50.133,Z -64.403,A -90.000,B 90.000,C 0.000} C_DIS
LIN {X 88.942,Y -50.133,Z -64.326,A -90.000,B 90.000,C 0.000} C_DIS
LIN {X 88.807,Y -50.125,Z -64.232,A -90.000,B 90.000,C 0.000} C_DIS
LIN {X 88.713,Y -50.120,Z -64.165,A -90.000,B 90.000,C 0.000} C_DIS
LIN {X 88.576,Y -50.107,Z -64.065,A -90.000,B 90.000,C 0.000} C_DIS
LIN {X 88.430,Y -50.105,Z -63.951,A -90.000,B 90.000,C 0.000} C_DIS
LIN {X 88.310,Y -50.104,Z -63.850,A -90.000,B 90.000,C 0.000} C_DIS
LIN {X 88.154,Y -50.106,Z -63.706,A -90.000,B 90.000,C 0.000} C_DIS
LIN {X 88.099,Y -50.109,Z -63.651,A -90.000,B 90.000,C 0.000} C_DIS
LIN {X 87.882,Y -50.100,Z -63.419,A -90.000,B 90.000,C 0.000} C_DIS
LIN {X 87.791,Y -50.089,Z -63.314,A -90.000,B 90.000,C 0.000} C_DIS
LIN {X 87.686,Y -50.079,Z -63.183,A -90.000,B 90.000,C 0.000} C_DIS
LIN {X 87.569,Y -50.056,Z -63.014,A -90.000,B 90.000,C 0.000} C_DIS
LIN {X 87.522,Y -50.049,Z -62.940,A -90.000,B 90.000,C 0.000} C_DIS
LIN {X 87.438,Y -50.025,Z -62.797,A -90.000,B 90.000,C 0.000} C_DIS
LIN {X 87.299,Y -49.989,Z -62.543,A -90.000,B 90.000,C 0.000} C_DIS
LIN {X 87.189,Y -49.957,Z -62.322,A -90.000,B 90.000,C 0.000} C_DIS
LIN {X 87.107,Y -49.937,Z -62.132,A -90.000,B 90.000,C 0.000} C_DIS
LIN {X 87.008,Y -49.912,Z -61.870,A -90.000,B 90.000,C 0.000} C_DIS
LIN {X 86.988,Y -49.908,Z -61.813,A -90.000,B 90.000,C 0.000} C_DIS
LIN {X 86.908,Y -49.867,Z -61.532,A -90.000,B 90.000,C 0.000} C_DIS
LIN {X 86.865,Y -49.835,Z -61.358,A -90.000,B 90.000,C 0.000} C_DIS
LIN {X 86.842,Y -49.816,Z -61.248,A -90.000,B 90.000,C 0.000} C_DIS
LIN {X 86.818,Y -49.796,Z -61.118,A -90.000,B 90.000,C 0.000} C_DIS
LIN {X 86.804,Y -49.781,Z -61.028,A -90.000,B 90.000,C 0.000} C_DIS
LIN {X 86.794,Y -49.764,Z -60.936,A -90.000,B 90.000,C 0.000} C_DIS
LIN {X 86.786,Y -49.745,Z -60.829,A -90.000,B 90.000,C 0.000} C_DIS
LIN {X 86.775,Y -49.716,Z -60.654,A -90.000,B 90.000,C 0.000} C_DIS
LIN {X 86.775,Y -49.661,Z -60.434,A -90.000,B 90.000,C 0.000} C_DIS
LIN {X 86.776,Y -49.637,Z -60.334,A -90.000,B 90.000,C 0.000} C_DIS
LIN {X 86.788,Y -49.600,Z -60.182,A -90.000,B 90.000,C 0.000} C_DIS
LIN {X 86.824,Y -49.510,Z -59.834,A -90.000,B 90.000,C 0.000} C_DIS
LIN {X 86.852,Y -49.464,Z -59.636,A -90.000,B 90.000,C 0.000} C_DIS
LIN {X 86.886,Y -49.427,Z -59.449,A -90.000,B 90.000,C 0.000} C_DIS
LIN {X 86.941,Y -49.377,Z -59.181,A -90.000,B 90.000,C 0.000} C_DIS
LIN {X 87.006,Y -49.327,Z -58.944,A -90.000,B 90.000,C 0.000} C_DIS
LIN {X 87.038,Y -49.308,Z -58.846,A -90.000,B 90.000,C 0.000} C_DIS
LIN {X 87.067,Y -49.304,Z -58.757,A -90.000,B 90.000,C 0.000} C_DIS
LIN {X 87.157,Y -49.263,Z -58.505,A -90.000,B 90.000,C 0.000} C_DIS
LIN {X 87.220,Y -49.241,Z -58.348,A -90.000,B 90.000,C 0.000} C_DIS
LIN {X 87.317,Y -49.214,Z -58.130,A -90.000,B 90.000,C 0.000} C_DIS
LIN {X 87.418,Y -49.200,Z -57.933,A -90.000,B 90.000,C 0.000} C_DIS
LIN {X 87.487,Y -49.197,Z -57.813,A -90.000,B 90.000,C 0.000} C_DIS
LIN {X 87.522,Y -49.198,Z -57.756,A -90.000,B 90.000,C 0.000} C_DIS
LIN {X 87.593,Y -49.205,Z -57.648,A -90.000,B 90.000,C 0.000} C_DIS
LIN {X 87.629,Y -49.211,Z -57.597,A -90.000,B 90.000,C 0.000} C_DIS
LIN {X 87.665,Y -49.219,Z -57.549,A -90.000,B 90.000,C 0.000} C_DIS
LIN {X 87.739,Y -49.240,Z -57.458,A -90.000,B 90.000,C 0.000} C_DIS
LIN {X 87.777,Y -49.253,Z -57.416,A -90.000,B 90.000,C 0.000} C_DIS
LIN {X 87.852,Y -49.283,Z -57.337,A -90.000,B 90.000,C 0.000} C_DIS
LIN {X 87.890,Y -49.301,Z -57.301,A -90.000,B 90.000,C 0.000} C_DIS
LIN {X 87.968,Y -49.341,Z -57.234,A -90.000,B 90.000,C 0.000} C_DIS
LIN {X 88.046,Y -49.385,Z -57.175,A -90.000,B 90.000,C 0.000} C_DIS
LIN {X 88.126,Y -49.431,Z -57.124,A -90.000,B 90.000,C 0.000} C_DIS
LIN {X 88.247,Y -49.505,Z -57.061,A -90.000,B 90.000,C 0.000} C_DIS
LIN {X 88.328,Y -49.557,Z -57.028,A -90.000,B 90.000,C 0.000} C_DIS
LIN {X 88.411,Y -49.612,Z -57.003,A -90.000,B 90.000,C 0.000} C_DIS
LIN {X 88.536,Y -49.698,Z -56.977,A -90.000,B 90.000,C 0.000} C_DIS
LIN {X 88.621,Y -49.757,Z -56.969,A -90.000,B 90.000,C 0.000} C_DIS
LIN {X 88.706,Y -49.820,Z -56.967,A -90.000,B 90.000,C 0.000} C_DIS
LIN {X 88.791,Y -49.885,Z -56.972,A -90.000,B 90.000,C 0.000} C_DIS
LIN {X 88.877,Y -49.952,Z -56.984,A -90.000,B 90.000,C 0.000} C_DIS
LIN {X 88.964,Y -50.021,Z -57.001,A -90.000,B 90.000,C 0.000} C_DIS
LIN {X 89.050,Y -50.091,Z -57.025,A -90.000,B 90.000,C 0.000} C_DIS
LIN {X 89.138,Y -50.161,Z -57.054,A -90.000,B 90.000,C 0.000} C_DIS
LIN {X 89.225,Y -50.232,Z -57.090,A -90.000,B 90.000,C 0.000} C_DIS
LIN {X 89.313,Y -50.302,Z -57.131,A -90.000,B 90.000,C 0.000} C_DIS
LIN {X 89.400,Y -50.372,Z -57.178,A -90.000,B 90.000,C 0.000} C_DIS
LIN {X 89.488,Y -50.441,Z -57.230,A -90.000,B 90.000,C 0.000} C_DIS
LIN {X 89.576,Y -50.510,Z -57.288,A -90.000,B 90.000,C 0.000} C_DIS
LIN {X 89.708,Y -50.618,Z -57.384,A -90.000,B 90.000,C 0.000} C_DIS
LIN {X 89.796,Y -50.691,Z -57.454,A -90.000,B 90.000,C 0.000} C_DIS
LIN {X 89.883,Y -50.762,Z -57.529,A -90.000,B 90.000,C 0.000} C_DIS
LIN {X 89.971,Y -50.832,Z -57.609,A -90.000,B 90.000,C 0.000} C_DIS
LIN {X 90.058,Y -50.899,Z -57.693,A -90.000,B 90.000,C 0.000} C_DIS
LIN {X 90.145,Y -50.963,Z -57.782,A -90.000,B 90.000,C 0.000} C_DIS
LIN {X 90.231,Y -51.023,Z -57.875,A -90.000,B 90.000,C 0.000} C_DIS
LIN {X 90.317,Y -51.080,Z -57.972,A -90.000,B 90.000,C 0.000} C_DIS
LIN {X 90.402,Y -51.133,Z -58.073,A -90.000,B 90.000,C 0.000} C_DIS
LIN {X 90.487,Y -51.182,Z -58.178,A -90.000,B 90.000,C 0.000} C_DIS
LIN {X 90.571,Y -51.226,Z -58.287,A -90.000,B 90.000,C 0.000} C_DIS
LIN {X 90.654,Y -51.267,Z -58.399,A -90.000,B 90.000,C 0.000} C_DIS
LIN {X 90.737,Y -51.303,Z -58.515,A -90.000,B 90.000,C 0.000} C_DIS
LIN {X 90.819,Y -51.335,Z -58.634,A -90.000,B 90.000,C 0.000} C_DIS
LIN {X 90.900,Y -51.362,Z -58.756,A -90.000,B 90.000,C 0.000} C_DIS
LIN {X 91.059,Y -51.412,Z -59.009,A -90.000,B 90.000,C 0.000} C_DIS
LIN {X 91.214,Y -51.459,Z -59.274,A -90.000,B 90.000,C 0.000} C_DIS
LIN {X 91.365,Y -51.494,Z -59.548,A -90.000,B 90.000,C 0.000} C_DIS
LIN {X 91.438,Y -51.506,Z -59.689,A -90.000,B 90.000,C 0.000} C_DIS
LIN {X 91.510,Y -51.512,Z -59.832,A -90.000,B 90.000,C 0.000} C_DIS
LIN {X 91.581,Y -51.513,Z -59.976,A -90.000,B 90.000,C 0.000} C_DIS
LIN {X 91.650,Y -51.508,Z -60.123,A -90.000,B 90.000,C 0.000} C_DIS
LIN {X 91.718,Y -51.499,Z -60.271,A -90.000,B 90.000,C 0.000} C_DIS
LIN {X 91.849,Y -51.466,Z -60.572,A -90.000,B 90.000,C 0.000} C_DIS
LIN {X 91.973,Y -51.433,Z -60.878,A -90.000,B 90.000,C 0.000} C_DIS
LIN {X 92.090,Y -51.395,Z -61.187,A -90.000,B 90.000,C 0.000} C_DIS
LIN {X 92.145,Y -51.371,Z -61.343,A -90.000,B 90.000,C 0.000} C_DIS
LIN {X 92.199,Y -51.340,Z -61.500,A -90.000,B 90.000,C 0.000} C_DIS
LIN {X 92.251,Y -51.303,Z -61.657,A -90.000,B 90.000,C 0.000} C_DIS
LIN {X 92.300,Y -51.260,Z -61.814,A -90.000,B 90.000,C 0.000} C_DIS
LIN {X 92.393,Y -51.161,Z -62.129,A -90.000,B 90.000,C 0.000} C_DIS
LIN {X 92.476,Y -51.055,Z -62.444,A -90.000,B 90.000,C 0.000} C_DIS
LIN {X 92.515,Y -51.001,Z -62.601,A -90.000,B 90.000,C 0.000} C_DIS
LIN {X 92.584,Y -50.903,Z -62.913,A -90.000,B 90.000,C 0.000} C_DIS
LIN {X 92.615,Y -50.849,Z -63.067,A -90.000,B 90.000,C 0.000} C_DIS
LIN {X 92.643,Y -50.792,Z -63.221,A -90.000,B 90.000,C 0.000} C_DIS
LIN {X 92.669,Y -50.732,Z -63.374,A -90.000,B 90.000,C 0.000} C_DIS
LIN {X 92.712,Y -50.608,Z -63.676,A -90.000,B 90.000,C 0.000} C_DIS
LIN {X 92.729,Y -50.548,Z -63.825,A -90.000,B 90.000,C 0.000} C_DIS
LIN {X 92.744,Y -50.494,Z -63.972,A -90.000,B 90.000,C 0.000} C_DIS
LIN {X 92.764,Y -50.396,Z -64.261,A -90.000,B 90.000,C 0.000} C_DIS
LIN {X 92.769,Y -50.348,Z -64.402,A -90.000,B 90.000,C 0.000} C_DIS
LIN {X 92.770,Y -50.251,Z -64.678,A -90.000,B 90.000,C 0.000} C_DIS
LIN {X 92.759,Y -50.151,Z -64.945,A -90.000,B 90.000,C 0.000} C_DIS
LIN {X 92.748,Y -50.100,Z -65.074,A -90.000,B 90.000,C 0.000} C_DIS
LIN {X 92.734,Y -50.053,Z -65.200,A -90.000,B 90.000,C 0.000} C_DIS
LIN {X 92.716,Y -50.011,Z -65.324,A -90.000,B 90.000,C 0.000} C_DIS
LIN {X 92.695,Y -49.968,Z -65.444,A -90.000,B 90.000,C 0.000} C_DIS
LIN {X 92.670,Y -49.924,Z -65.561,A -90.000,B 90.000,C 0.000} C_DIS
LIN {X 92.642,Y -49.879,Z -65.675,A -90.000,B 90.000,C 0.000} C_DIS
LIN {X 92.610,Y -49.832,Z -65.785,A -90.000,B 90.000,C 0.000} C_DIS
LIN {X 92.574,Y -49.784,Z -65.891,A -90.000,B 90.000,C 0.000} C_DIS
LIN {X 92.534,Y -49.736,Z -65.994,A -90.000,B 90.000,C 0.000} C_DIS
LIN {X 92.491,Y -49.690,Z -66.092,A -90.000,B 90.000,C 0.000} C_DIS
LIN {X 92.443,Y -49.646,Z -66.187,A -90.000,B 90.000,C 0.000} C_DIS
LIN {X 92.392,Y -49.604,Z -66.277,A -90.000,B 90.000,C 0.000} C_DIS
LIN {X 92.337,Y -49.564,Z -66.363,A -90.000,B 90.000,C 0.000} C_DIS
LIN {X 92.277,Y -49.530,Z -66.445,A -90.000,B 90.000,C 0.000} C_DIS
LIN {X 92.213,Y -49.498,Z -66.521,A -90.000,B 90.000,C 0.000} C_DIS
LIN {X 92.145,Y -49.468,Z -66.593,A -90.000,B 90.000,C 0.000} C_DIS
LIN {X 92.073,Y -49.439,Z -66.661,A -90.000,B 90.000,C 0.000} C_DIS
LIN {X 91.997,Y -49.413,Z -66.723,A -90.000,B 90.000,C 0.000} C_DIS
LIN {X 91.916,Y -49.389,Z -66.780,A -90.000,B 90.000,C 0.000} C_DIS
LIN {X 91.830,Y -49.367,Z -66.831,A -90.000,B 90.000,C 0.000} C_DIS
LIN {X 91.694,Y -49.337,Z -66.898,A -90.000,B 90.000,C 0.000} C_DIS
LIN {X 91.597,Y -49.321,Z -66.936,A -90.000,B 90.000,C 0.000} C_DIS
LIN {X 91.495,Y -49.306,Z -66.968,A -90.000,B 90.000,C 0.000} C_DIS
LIN {X 91.335,Y -49.289,Z -67.004,A -90.000,B 90.000,C 0.000} C_DIS
LIN {X 91.221,Y -49.280,Z -67.021,A -90.000,B 90.000,C 0.000} C_DIS
LIN {X 91.103,Y -49.274,Z -67.032,A -90.000,B 90.000,C 0.000} C_DIS
LIN {X 90.917,Y -49.275,Z -67.035,A -90.000,B 90.000,C 0.000} C_DIS
LIN {X 90.719,Y -49.280,Z -67.024,A -90.000,B 90.000,C 0.000} C_DIS
LIN {X 90.581,Y -49.282,Z -67.008,A -90.000,B 90.000,C 0.000} C_DIS
LIN {X 90.438,Y -49.284,Z -66.985,A -90.000,B 90.000,C 0.000} C_DIS
LIN {X 90.213,Y -49.284,Z -66.937,A -90.000,B 90.000,C 0.000} C_DIS
LIN {X 90.056,Y -49.287,Z -66.896,A -90.000,B 90.000,C 0.000} C_DIS
LIN {X 89.895,Y -49.293,Z -66.848,A -90.000,B 90.000,C 0.000} C_DIS
LIN {X 89.728,Y -49.300,Z -66.792,A -90.000,B 90.000,C 0.000} C_DIS
LIN {X 89.555,Y -49.310,Z -66.728,A -90.000,B 90.000,C 0.000} C_DIS
LIN {X 89.467,Y -49.308,Z -66.693,A -90.000,B 90.000,C 0.000} C_DIS
LIN {X 89.386,Y -49.315,Z -66.661,A -90.000,B 90.000,C 0.000} C_DIS
LIN {X 89.261,Y -49.324,Z -66.608,A -90.000,B 90.000,C 0.000} C_DIS
LIN {X 89.129,Y -49.334,Z -66.547,A -90.000,B 90.000,C 0.000} C_DIS
LIN {X 88.835,Y -49.345,Z -66.393,A -90.000,B 90.000,C 0.000} C_DIS
LIN {X 88.144,Y -49.365,Z -66.003,A -90.000,B 90.000,C 0.000} C_DIS
LIN {X 88.024,Y -49.370,Z -65.932,A -90.000,B 90.000,C 0.000} C_DIS
LIN {X 87.880,Y -49.370,Z -65.840,A -90.000,B 90.000,C 0.000} C_DIS
LIN {X 87.757,Y -49.371,Z -65.759,A -90.000,B 90.000,C 0.000} C_DIS
LIN {X 87.486,Y -49.353,Z -65.563,A -90.000,B 90.000,C 0.000} C_DIS
LIN {X 87.214,Y -49.333,Z -65.340,A -90.000,B 90.000,C 0.000} C_DIS
LIN {X 87.127,Y -49.328,Z -65.264,A -90.000,B 90.000,C 0.000} C_DIS
LIN {X 87.002,Y -49.324,Z -65.148,A -90.000,B 90.000,C 0.000} C_DIS
LIN {X 86.876,Y -49.320,Z -65.028,A -90.000,B 90.000,C 0.000} C_DIS
LIN {X 86.665,Y -49.308,Z -64.803,A -90.000,B 90.000,C 0.000} C_DIS
LIN {X 86.665,Y -60.000,Z -64.803,A -90.000,B 90.000,C 0.000} C_DIS
LIN {X 98.892,Y -60.000,Z -48.885,A -90.000,B 90.000,C 0.000} C_DIS
LIN {X 98.892,Y -49.308,Z -48.885,A -90.000,B 90.000,C 0.000} C_DIS
LIN {X 98.952,Y -49.332,Z -48.897,A -90.000,B 90.000,C 0.000} C_DIS
LIN {X 99.118,Y -49.389,Z -48.936,A -90.000,B 90.000,C 0.000} C_DIS
LIN {X 99.256,Y -49.439,Z -48.972,A -90.000,B 90.000,C 0.000} C_DIS
LIN {X 99.351,Y -49.475,Z -48.999,A -90.000,B 90.000,C 0.000} C_DIS
LIN {X 99.554,Y -49.538,Z -49.064,A -90.000,B 90.000,C 0.000} C_DIS
LIN {X 99.780,Y -49.600,Z -49.150,A -90.000,B 90.000,C 0.000} C_DIS
LIN {X 99.915,Y -49.638,Z -49.204,A -90.000,B 90.000,C 0.000} C_DIS
LIN {X 100.096,Y -49.686,Z -49.290,A -90.000,B 90.000,C 0.000} C_DIS
LIN {X 100.233,Y -49.717,Z -49.361,A -90.000,B 90.000,C 0.000} C_DIS
LIN {X 100.464,Y -49.765,Z -49.494,A -90.000,B 90.000,C 0.000} C_DIS
LIN {X 100.716,Y -49.815,Z -49.651,A -90.000,B 90.000,C 0.000} C_DIS
LIN {X 100.796,Y -49.831,Z -49.704,A -90.000,B 90.000,C 0.000} C_DIS
LIN {X 100.978,Y -49.863,Z -49.834,A -90.000,B 90.000,C 0.000} C_DIS
LIN {X 101.186,Y -49.886,Z -49.999,A -90.000,B 90.000,C 0.000} C_DIS
LIN {X 101.401,Y -49.899,Z -50.194,A -90.000,B 90.000,C 0.000} C_DIS
LIN {X 101.484,Y -49.899,Z -50.277,A -90.000,B 90.000,C 0.000} C_DIS
LIN {X 101.588,Y -49.901,Z -50.386,A -90.000,B 90.000,C 0.000} C_DIS
LIN {X 101.700,Y -49.895,Z -50.509,A -90.000,B 90.000,C 0.000} C_DIS
LIN {X 101.773,Y -49.891,Z -50.595,A -90.000,B 90.000,C 0.000} C_DIS
LIN {X 102.054,Y -49.853,Z -50.939,A -90.000,B 90.000,C 0.000} C_DIS
LIN {X 102.191,Y -49.822,Z -51.120,A -90.000,B 90.000,C 0.000} C_DIS
LIN {X 102.333,Y -49.789,Z -51.322,A -90.000,B 90.000,C 0.000} C_DIS
LIN {X 102.494,Y -49.742,Z -51.580,A -90.000,B 90.000,C 0.000} C_DIS
LIN {X 102.621,Y -49.693,Z -51.819,A -90.000,B 90.000,C 0.000} C_DIS
LIN {X 102.697,Y -49.644,Z -51.985,A -90.000,B 90.000,C 0.000} C_DIS
LIN {X 102.774,Y -49.593,Z -52.169,A -90.000,B 90.000,C 0.000} C_DIS
LIN {X 102.793,Y -49.580,Z -52.221,A -90.000,B 90.000,C 0.000} C_DIS
LIN {X 102.912,Y -49.503,Z -52.534,A -90.000,B 90.000,C 0.000} C_DIS
LIN {X 102.954,Y -49.475,Z -52.658,A -90.000,B 90.000,C 0.000} C_DIS
LIN {X 103.028,Y -49.422,Z -52.892,A -90.000,B 90.000,C 0.000} C_DIS
LIN {X 103.083,Y -49.351,Z -53.127,A -90.000,B 90.000,C 0.000} C_DIS
LIN {X 103.120,Y -49.308,Z -53.305,A -90.000,B 90.000,C 0.000} C_DIS
LIN {X 103.059,Y -49.308,Z -53.664,A -90.000,B 90.000,C 0.000} C_DIS
LIN {X 102.974,Y -49.308,Z -54.078,A -90.000,B 90.000,C 0.000} C_DIS
LIN {X 102.866,Y -49.308,Z -54.511,A -90.000,B 90.000,C 0.000} C_DIS
LIN {X 102.682,Y -49.308,Z -55.021,A -90.000,B 90.000,C 0.000} C_DIS
LIN {X 102.608,Y -49.308,Z -55.285,A -90.000,B 90.000,C 0.000} C_DIS
LIN {X 102.383,Y -49.308,Z -55.942,A -90.000,B 90.000,C 0.000} C_DIS
LIN {X 102.146,Y -49.308,Z -56.762,A -90.000,B 90.000,C 0.000} C_DIS
LIN {X 102.025,Y -49.308,Z -57.189,A -90.000,B 90.000,C 0.000} C_DIS
LIN {X 101.895,Y -49.308,Z -57.515,A -90.000,B 90.000,C 0.000} C_DIS
LIN {X 101.243,Y -49.308,Z -59.064,A -90.000,B 90.000,C 0.000} C_DIS
LIN {X 100.896,Y -49.308,Z -59.914,A -90.000,B 90.000,C 0.000} C_DIS
LIN {X 100.682,Y -49.308,Z -60.287,A -90.000,B 90.000,C 0.000} C_DIS
LIN {X 99.946,Y -49.308,Z -61.572,A -90.000,B 90.000,C 0.000} C_DIS
LIN {X 99.572,Y -49.308,Z -62.227,A -90.000,B 90.000,C 0.000} C_DIS
LIN {X 99.518,Y -49.308,Z -62.316,A -90.000,B 90.000,C 0.000} C_DIS
LIN {X 99.417,Y -49.308,Z -62.472,A -90.000,B 90.000,C 0.000} C_DIS
LIN {X 99.154,Y -49.308,Z -62.817,A -90.000,B 90.000,C 0.000} C_DIS
LIN {X 97.806,Y -49.308,Z -64.413,A -90.000,B 90.000,C 0.000} C_DIS
LIN {X 97.593,Y -49.308,Z -64.651,A -90.000,B 90.000,C 0.000} C_DIS
LIN {X 97.532,Y -49.308,Z -64.715,A -90.000,B 90.000,C 0.000} C_DIS
LIN {X 97.285,Y -49.308,Z -64.917,A -90.000,B 90.000,C 0.000} C_DIS
LIN {X 96.193,Y -49.308,Z -65.689,A -90.000,B 90.000,C 0.000} C_DIS
LIN {X 95.917,Y -49.308,Z -65.850,A -90.000,B 90.000,C 0.000} C_DIS
LIN {X 94.825,Y -49.308,Z -66.418,A -90.000,B 90.000,C 0.000} C_DIS
LIN {X 94.735,Y -49.308,Z -66.469,A -90.000,B 90.000,C 0.000} C_DIS
LIN {X 94.425,Y -49.308,Z -66.591,A -90.000,B 90.000,C 0.000} C_DIS
LIN {X 94.314,Y -49.308,Z -66.632,A -90.000,B 90.000,C 0.000} C_DIS
LIN {X 93.366,Y -49.308,Z -66.866,A -90.000,B 90.000,C 0.000} C_DIS
LIN {X 93.054,Y -49.308,Z -66.934,A -90.000,B 90.000,C 0.000} C_DIS
LIN {X 92.735,Y -49.308,Z -66.953,A -90.000,B 90.000,C 0.000} C_DIS
LIN {X 92.293,Y -49.308,Z -66.972,A -90.000,B 90.000,C 0.000} C_DIS
LIN {X 91.836,Y -49.308,Z -66.963,A -90.000,B 90.000,C 0.000} C_DIS
LIN {X 91.353,Y -49.308,Z -66.942,A -90.000,B 90.000,C 0.000} C_DIS
LIN {X 90.907,Y -49.308,Z -66.963,A -90.000,B 90.000,C 0.000} C_DIS
LIN {X 90.589,Y -49.308,Z -66.932,A -90.000,B 90.000,C 0.000} C_DIS
LIN {X 90.467,Y -49.308,Z -66.910,A -90.000,B 90.000,C 0.000} C_DIS
LIN {X 90.195,Y -49.308,Z -66.857,A -90.000,B 90.000,C 0.000} C_DIS
LIN {X 90.014,Y -49.308,Z -66.818,A -90.000,B 90.000,C 0.000} C_DIS
LIN {X 89.451,Y -49.308,Z -66.690,A -90.000,B 90.000,C 0.000} C_DIS
LIN {X 89.421,Y -49.308,Z -66.687,A -90.000,B 90.000,C 0.000} C_DIS
LIN {X 89.112,Y -49.308,Z -66.606,A -90.000,B 90.000,C 0.000} C_DIS
LIN {X 89.054,Y -49.308,Z -66.584,A -90.000,B 90.000,C 0.000} C_DIS
LIN {X 88.811,Y -49.308,Z -66.478,A -90.000,B 90.000,C 0.000} C_DIS
LIN {X 88.514,Y -49.308,Z -66.335,A -90.000,B 90.000,C 0.000} C_DIS
LIN {X 87.954,Y -49.308,Z -66.030,A -90.000,B 90.000,C 0.000} C_DIS
LIN {X 87.685,Y -49.308,Z -65.858,A -90.000,B 90.000,C 0.000} C_DIS
LIN {X 87.458,Y -49.308,Z -65.658,A -90.000,B 90.000,C 0.000} C_DIS
LIN {X 87.445,Y -49.308,Z -65.647,A -90.000,B 90.000,C 0.000} C_DIS
LIN {X 87.408,Y -49.308,Z -65.602,A -90.000,B 90.000,C 0.000} C_DIS
LIN {X 86.854,Y -49.308,Z -65.036,A -90.000,B 90.000,C 0.000} C_DIS
LIN {X 86.689,Y -49.308,Z -64.837,A -90.000,B 90.000,C 0.000} C_DIS
LIN {X 86.650,Y -49.308,Z -64.783,A -90.000,B 90.000,C 0.000} C_DIS
LIN {X 86.518,Y -49.308,Z -64.560,A -90.000,B 90.000,C 0.000} C_DIS
LIN {X 86.487,Y -49.308,Z -64.501,A -90.000,B 90.000,C 0.000} C_DIS
LIN {X 86.391,Y -49.308,Z -64.261,A -90.000,B 90.000,C 0.000} C_DIS
LIN {X 86.369,Y -49.308,Z -64.198,A -90.000,B 90.000,C 0.000} C_DIS
LIN {X 86.271,Y -49.308,Z -63.764,A -90.000,B 90.000,C 0.000} C_DIS
LIN {X 86.088,Y -49.308,Z -62.858,A -90.000,B 90.000,C 0.000} C_DIS
LIN {X 86.068,Y -49.308,Z -62.507,A -90.000,B 90.000,C 0.000} C_DIS
LIN {X 86.077,Y -49.308,Z -62.127,A -90.000,B 90.000,C 0.000} C_DIS
LIN {X 86.094,Y -49.308,Z -61.748,A -90.000,B 90.000,C 0.000} C_DIS
LIN {X 86.219,Y -49.308,Z -60.982,A -90.000,B 90.000,C 0.000} C_DIS
LIN {X 86.301,Y -49.308,Z -60.625,A -90.000,B 90.000,C 0.000} C_DIS
LIN {X 86.382,Y -49.308,Z -60.301,A -90.000,B 90.000,C 0.000} C_DIS
LIN {X 86.521,Y -49.308,Z -59.923,A -90.000,B 90.000,C 0.000} C_DIS
LIN {X 86.775,Y -49.308,Z -59.351,A -90.000,B 90.000,C 0.000} C_DIS
LIN {X 86.959,Y -49.308,Z -58.993,A -90.000,B 90.000,C 0.000} C_DIS
LIN {X 87.533,Y -49.308,Z -57.919,A -90.000,B 90.000,C 0.000} C_DIS
LIN {X 87.919,Y -49.308,Z -57.280,A -90.000,B 90.000,C 0.000} C_DIS
LIN {X 88.064,Y -49.308,Z -57.063,A -90.000,B 90.000,C 0.000} C_DIS
LIN {X 88.162,Y -49.308,Z -56.921,A -90.000,B 90.000,C 0.000} C_DIS
LIN {X 88.331,Y -49.308,Z -56.722,A -90.000,B 90.000,C 0.000} C_DIS
LIN {X 88.445,Y -49.308,Z -56.592,A -90.000,B 90.000,C 0.000} C_DIS
LIN {X 89.379,Y -49.308,Z -55.576,A -90.000,B 90.000,C 0.000} C_DIS
LIN {X 90.245,Y -49.308,Z -54.667,A -90.000,B 90.000,C 0.000} C_DIS
LIN {X 90.357,Y -49.308,Z -54.554,A -90.000,B 90.000,C 0.000} C_DIS
LIN {X 90.566,Y -49.308,Z -54.358,A -90.000,B 90.000,C 0.000} C_DIS
LIN {X 92.731,Y -49.308,Z -52.546,A -90.000,B 90.000,C 0.000} C_DIS
LIN {X 92.803,Y -49.308,Z -52.488,A -90.000,B 90.000,C 0.000} C_DIS
LIN {X 93.084,Y -49.308,Z -52.278,A -90.000,B 90.000,C 0.000} C_DIS
LIN {X 93.639,Y -49.308,Z -51.880,A -90.000,B 90.000,C 0.000} C_DIS
LIN {X 95.430,Y -49.308,Z -50.650,A -90.000,B 90.000,C 0.000} C_DIS
LIN {X 95.880,Y -49.308,Z -50.377,A -90.000,B 90.000,C 0.000} C_DIS
LIN {X 97.279,Y -49.308,Z -49.603,A -90.000,B 90.000,C 0.000} C_DIS
LIN {X 97.637,Y -49.308,Z -49.418,A -90.000,B 90.000,C 0.000} C_DIS
LIN {X 98.112,Y -49.308,Z -49.187,A -90.000,B 90.000,C 0.000} C_DIS
LIN {X 98.648,Y -49.308,Z -48.972,A -90.000,B 90.000,C 0.000} C_DIS
LIN {X 99.005,Y -49.308,Z -48.845,A -90.000,B 90.000,C 0.000} C_DIS
LIN {X 99.727,Y -49.308,Z -48.635,A -90.000,B 90.000,C 0.000} C_DIS
LIN {X 100.071,Y -49.308,Z -48.563,A -90.000,B 90.000,C 0.000} C_DIS
LIN {X 100.622,Y -49.308,Z -48.486,A -90.000,B 90.000,C 0.000} C_DIS
LIN {X 100.941,Y -49.308,Z -48.464,A -90.000,B 90.000,C 0.000} C_DIS
LIN {X 100.964,Y -49.308,Z -48.464,A -90.000,B 90.000,C 0.000} C_DIS
LIN {X 101.282,Y -49.308,Z -48.491,A -90.000,B 90.000,C 0.000} C_DIS
LIN {X 101.432,Y -49.308,Z -48.514,A -90.000,B 90.000,C 0.000} C_DIS
LIN {X 101.742,Y -49.308,Z -48.590,A -90.000,B 90.000,C 0.000} C_DIS
LIN {X 101.867,Y -49.308,Z -48.625,A -90.000,B 90.000,C 0.000} C_DIS
LIN {X 102.173,Y -49.308,Z -48.753,A -90.000,B 90.000,C 0.000} C_DIS
LIN {X 102.326,Y -49.308,Z -48.843,A -90.000,B 90.000,C 0.000} C_DIS
LIN {X 102.437,Y -49.308,Z -48.916,A -90.000,B 90.000,C 0.000} C_DIS
LIN {X 102.559,Y -49.308,Z -49.001,A -90.000,B 90.000,C 0.000} C_DIS
LIN {X 102.761,Y -49.308,Z -49.198,A -90.000,B 90.000,C 0.000} C_DIS
LIN {X 102.894,Y -49.308,Z -49.373,A -90.000,B 90.000,C 0.000} C_DIS
LIN {X 103.060,Y -49.308,Z -49.646,A -90.000,B 90.000,C 0.000} C_DIS
LIN {X 103.175,Y -49.308,Z -49.925,A -90.000,B 90.000,C 0.000} C_DIS
LIN {X 103.317,Y -49.308,Z -50.347,A -90.000,B 90.000,C 0.000} C_DIS
LIN {X 103.392,Y -49.308,Z -50.663,A -90.000,B 90.000,C 0.000} C_DIS
LIN {X 103.419,Y -49.308,Z -50.985,A -90.000,B 90.000,C 0.000} C_DIS
LIN {X 103.419,Y -49.308,Z -51.053,A -90.000,B 90.000,C 0.000} C_DIS
LIN {X 103.334,Y -49.308,Z -51.883,A -90.000,B 90.000,C 0.000} C_DIS
LIN {X 103.305,Y -49.308,Z -52.091,A -90.000,B 90.000,C 0.000} C_DIS
LIN {X 103.290,Y -49.308,Z -52.300,A -90.000,B 90.000,C 0.000} C_DIS
LIN {X 103.256,Y -49.308,Z -52.649,A -90.000,B 90.000,C 0.000} C_DIS
LIN {X 103.157,Y -49.308,Z -53.081,A -90.000,B 90.000,C 0.000} C_DIS
LIN {X 103.120,Y -49.308,Z -53.305,A -90.000,B 90.000,C 0.000} C_DIS
LIN {X 103.023,Y -49.303,Z -53.929,A -90.000,B 90.000,C 0.000} C_DIS
LIN {X 103.001,Y -49.297,Z -54.085,A -90.000,B 90.000,C 0.000} C_DIS
LIN {X 102.976,Y -49.291,Z -54.240,A -90.000,B 90.000,C 0.000} C_DIS
LIN {X 102.927,Y -49.267,Z -54.551,A -90.000,B 90.000,C 0.000} C_DIS
LIN {X 102.859,Y -49.243,Z -54.855,A -90.000,B 90.000,C 0.000} C_DIS
LIN {X 102.820,Y -49.228,Z -55.045,A -90.000,B 90.000,C 0.000} C_DIS
LIN {X 102.787,Y -49.198,Z -55.318,A -90.000,B 90.000,C 0.000} C_DIS
LIN {X 102.719,Y -49.148,Z -55.781,A -90.000,B 90.000,C 0.000} C_DIS
LIN {X 102.690,Y -49.122,Z -56.014,A -90.000,B 90.000,C 0.000} C_DIS
LIN {X 102.672,Y -49.097,Z -56.249,A -90.000,B 90.000,C 0.000} C_DIS
LIN {X 102.644,Y -49.045,Z -56.722,A -90.000,B 90.000,C 0.000} C_DIS
LIN {X 102.622,Y -48.985,Z -57.276,A -90.000,B 90.000,C 0.000} C_DIS
LIN {X 102.585,Y -48.943,Z -57.663,A -90.000,B 90.000,C 0.000} C_DIS
LIN {X 102.509,Y -48.876,Z -58.276,A -90.000,B 90.000,C 0.000} C_DIS
LIN {X 102.427,Y -48.810,Z -58.888,A -90.000,B 90.000,C 0.000} C_DIS
LIN {X 102.342,Y -48.743,Z -59.498,A -90.000,B 90.000,C 0.000} C_DIS
LIN {X 102.250,Y -48.676,Z -60.109,A -90.000,B 90.000,C 0.000} C_DIS
LIN {X 102.178,Y -48.634,Z -60.485,A -90.000,B 90.000,C 0.000} C_DIS
LIN {X 102.119,Y -48.607,Z -60.726,A -90.000,B 90.000,C 0.000} C_DIS
LIN {X 102.031,Y -48.577,Z -60.995,A -90.000,B 90.000,C 0.000} C_DIS
LIN {X 101.879,Y -48.528,Z -61.423,A -90.000,B 90.000,C 0.000} C_DIS
LIN {X 101.769,Y -48.495,Z -61.707,A -90.000,B 90.000,C 0.000} C_DIS
LIN {X 101.652,Y -48.462,Z -61.989,A -90.000,B 90.000,C 0.000} C_DIS
LIN {X 101.590,Y -48.445,Z -62.130,A -90.000,B 90.000,C 0.000} C_DIS
LIN {X 101.460,Y -48.411,Z -62.409,A -90.000,B 90.000,C 0.000} C_DIS
LIN {X 101.319,Y -48.378,Z -62.687,A -90.000,B 90.000,C 0.000} C_DIS
LIN {X 101.169,Y -48.344,Z -62.963,A -90.000,B 90.000,C 0.000} C_DIS
LIN {X 101.168,Y -48.344,Z -62.964,A -90.000,B 90.000,C 0.000} C_DIS
LIN {X 101.030,Y -48.344,Z -63.203,A -90.000,B 90.000,C 0.000} C_DIS
LIN {X 100.990,Y -48.345,Z -63.267,A -90.000,B 90.000,C 0.000} C_DIS
LIN {X 100.889,Y -48.342,Z -63.421,A -90.000,B 90.000,C 0.000} C_DIS
LIN {X 100.809,Y -48.343,Z -63.534,A -90.000,B 90.000,C 0.000} C_DIS
LIN {X 100.549,Y -48.350,Z -63.882,A -90.000,B 90.000,C 0.000} C_DIS
LIN {X 100.495,Y -48.353,Z -63.952,A -90.000,B 90.000,C 0.000} C_DIS
LIN {X 100.262,Y -48.368,Z -64.240,A -90.000,B 90.000,C 0.000} C_DIS
LIN {X 99.710,Y -48.392,Z -64.914,A -90.000,B 90.000,C 0.000} C_DIS
LIN {X 99.354,Y -48.403,Z -65.343,A -90.000,B 90.000,C 0.000} C_DIS
LIN {X 99.148,Y -48.399,Z -65.585,A -90.000,B 90.000,C 0.000} C_DIS
LIN {X 98.884,Y -48.390,Z -65.871,A -90.000,B 90.000,C 0.000} C_DIS
LIN {X 98.823,Y -48.389,Z -65.935,A -90.000,B 90.000,C 0.000} C_DIS
LIN {X 98.657,Y -48.392,Z -66.092,A -90.000,B 90.000,C 0.000} C_DIS
LIN {X 98.414,Y -48.405,Z -66.299,A -90.000,B 90.000,C 0.000} C_DIS
LIN {X 98.351,Y -48.410,Z -66.351,A -90.000,B 90.000,C 0.000} C_DIS
LIN {X 97.219,Y -48.447,Z -67.174,A -90.000,B 90.000,C 0.000} C_DIS
LIN {X 97.175,Y -48.450,Z -67.205,A -90.000,B 90.000,C 0.000} C_DIS
LIN {X 96.948,Y -48.466,Z -67.348,A -90.000,B 90.000,C 0.000} C_DIS
LIN {X 96.768,Y -48.471,Z -67.455,A -90.000,B 90.000,C 0.000} C_DIS
LIN {X 96.479,Y -48.477,Z -67.608,A -90.000,B 90.000,C 0.000} C_DIS
LIN {X 95.691,Y -48.485,Z -68.022,A -90.000,B 90.000,C 0.000} C_DIS
LIN {X 95.562,Y -48.485,Z -68.093,A -90.000,B 90.000,C 0.000} C_DIS
LIN {X 95.374,Y -48.482,Z -68.175,A -90.000,B 90.000,C 0.000} C_DIS
LIN {X 95.264,Y -48.481,Z -68.218,A -90.000,B 90.000,C 0.000} C_DIS
LIN {X 94.948,Y -48.476,Z -68.336,A -90.000,B 90.000,C 0.000} C_DIS
LIN {X 94.749,Y -48.478,Z -68.398,A -90.000,B 90.000,C 0.000} C_DIS
LIN {X 94.612,Y -48.482,Z -68.434,A -90.000,B 90.000,C 0.000} C_DIS
LIN {X 94.161,Y -48.506,Z -68.556,A -90.000,B 90.000,C 0.000} C_DIS
LIN {X 93.803,Y -48.502,Z -68.643,A -90.000,B 90.000,C 0.000} C_DIS
LIN {X 93.374,Y -48.497,Z -68.734,A -90.000,B 90.000,C 0.000} C_DIS
LIN {X 93.341,Y -48.497,Z -68.739,A -90.000,B 90.000,C 0.000} C_DIS
LIN {X 93.161,Y -48.502,Z -68.761,A -90.000,B 90.000,C 0.000} C_DIS
LIN {X 92.755,Y -48.519,Z -68.791,A -90.000,B 90.000,C 0.000} C_DIS
LIN {X 92.431,Y -48.521,Z -68.806,A -90.000,B 90.000,C 0.000} C_DIS
LIN {X 92.333,Y -48.518,Z -68.809,A -90.000,B 90.000,C 0.000} C_DIS
LIN {X 91.997,Y -48.522,Z -68.805,A -90.000,B 90.000,C 0.000} C_DIS
LIN {X 91.726,Y -48.526,Z -68.800,A -90.000,B 90.000,C 0.000} C_DIS
LIN {X 91.415,Y -48.532,Z -68.789,A -90.000,B 90.000,C 0.000} C_DIS
LIN {X 91.357,Y -48.531,Z -68.786,A -90.000,B 90.000,C 0.000} C_DIS
LIN {X 91.094,Y -48.517,Z -68.793,A -90.000,B 90.000,C 0.000} C_DIS
LIN {X 90.927,Y -48.502,Z -68.793,A -90.000,B 90.000,C 0.000} C_DIS
LIN {X 90.835,Y -48.495,Z -68.789,A -90.000,B 90.000,C 0.000} C_DIS
LIN {X 90.688,Y -48.489,Z -68.775,A -90.000,B 90.000,C 0.000} C_DIS
LIN {X 90.385,Y -48.471,Z -68.737,A -90.000,B 90.000,C 0.000} C_DIS
LIN {X 90.152,Y -48.461,Z -68.694,A -90.000,B 90.000,C 0.000} C_DIS
LIN {X 89.946,Y -48.454,Z -68.651,A -90.000,B 90.000,C 0.000} C_DIS
LIN {X 89.717,Y -48.458,Z -68.606,A -90.000,B 90.000,C 0.000} C_DIS
LIN {X 89.446,Y -48.464,Z -68.548,A -90.000,B 90.000,C 0.000} C_DIS
LIN {X 89.122,Y -48.460,Z -68.473,A -90.000,B 90.000,C 0.000} C_DIS
LIN {X 89.017,Y -48.451,Z -68.448,A -90.000,B 90.000,C 0.000} C_DIS
LIN {X 88.609,Y -48.425,Z -68.329,A -90.000,B 90.000,C 0.000} C_DIS
LIN {X 88.514,Y -48.421,Z -68.296,A -90.000,B 90.000,C 0.000} C_DIS
LIN {X 88.415,Y -48.418,Z -68.257,A -90.000,B 90.000,C 0.000} C_DIS
LIN {X 88.245,Y -48.416,Z -68.184,A -90.000,B 90.000,C 0.000} C_DIS
LIN {X 88.028,Y -48.425,Z -68.093,A -90.000,B 90.000,C 0.000} C_DIS
LIN {X 87.764,Y -48.430,Z -67.968,A -90.000,B 90.000,C 0.000} C_DIS
LIN {X 87.655,Y -48.425,Z -67.910,A -90.000,B 90.000,C 0.000} C_DIS
LIN {X 87.483,Y -48.420,Z -67.814,A -90.000,B 90.000,C 0.000} C_DIS
LIN {X 87.102,Y -48.399,Z -67.594,A -90.000,B 90.000,C 0.000} C_DIS
LIN {X 86.999,Y -48.395,Z -67.531,A -90.000,B 90.000,C 0.000} C_DIS
LIN {X 86.904,Y -48.393,Z -67.469,A -90.000,B 90.000,C 0.000} C_DIS
LIN {X 86.875,Y -48.393,Z -67.451,A -90.000,B 90.000,C 0.000} C_DIS
LIN {X 86.730,Y -48.393,Z -67.358,A -90.000,B 90.000,C 0.000} C_DIS
LIN {X 86.642,Y -48.394,Z -67.300,A -90.000,B 90.000,C 0.000} C_DIS
LIN {X 86.610,Y -48.393,Z -67.274,A -90.000,B 90.000,C 0.000} C_DIS
LIN {X 86.509,Y -48.391,Z -67.191,A -90.000,B 90.000,C 0.000} C_DIS
LIN {X 86.399,Y -48.391,Z -67.094,A -90.000,B 90.000,C 0.000} C_DIS
LIN {X 86.264,Y -48.379,Z -66.966,A -90.000,B 90.000,C 0.000} C_DIS
LIN {X 86.175,Y -48.373,Z -66.876,A -90.000,B 90.000,C 0.000} C_DIS
LIN {X 86.092,Y -48.369,Z -66.782,A -90.000,B 90.000,C 0.000} C_DIS
LIN {X 85.856,Y -48.353,Z -66.528,A -90.000,B 90.000,C 0.000} C_DIS
LIN {X 85.659,Y -48.351,Z -66.326,A -90.000,B 90.000,C 0.000} C_DIS
LIN {X 85.582,Y -48.344,Z -66.241,A -90.000,B 90.000,C 0.000} C_DIS
LIN {X 85.494,Y -48.339,Z -66.137,A -90.000,B 90.000,C 0.000} C_DIS
LIN {X 85.436,Y -48.336,Z -66.064,A -90.000,B 90.000,C 0.000} C_DIS
LIN {X 85.318,Y -48.318,Z -65.904,A -90.000,B 90.000,C 0.000} C_DIS
LIN {X 85.243,Y -48.309,Z -65.794,A -90.000,B 90.000,C 0.000} C_DIS
LIN {X 85.195,Y -48.298,Z -65.712,A -90.000,B 90.000,C 0.000} C_DIS
LIN {X 85.089,Y -48.277,Z -65.511,A -90.000,B 90.000,C 0.000} C_DIS
LIN {X 85.042,Y -48.265,Z -65.417,A -90.000,B 90.000,C 0.000} C_DIS
LIN {X 84.985,Y -48.252,Z -65.293,A -90.000,B 90.000,C 0.000} C_DIS
LIN {X 84.941,Y -48.243,Z -65.191,A -90.000,B 90.000,C 0.000} C_DIS
LIN {X 84.852,Y -48.230,Z -64.949,A -90.000,B 90.000,C 0.000} C_DIS
LIN {X 84.790,Y -48.218,Z -64.761,A -90.000,B 90.000,C 0.000} C_DIS
LIN {X 84.756,Y -48.213,Z -64.642,A -90.000,B 90.000,C 0.000} C_DIS
LIN {X 84.671,Y -48.212,Z -64.274,A -90.000,B 90.000,C 0.000} C_DIS
LIN {X 84.639,Y -48.200,Z -64.092,A -90.000,B 90.000,C 0.000} C_DIS
LIN {X 84.575,Y -48.178,Z -63.697,A -90.000,B 90.000,C 0.000} C_DIS
LIN {X 84.529,Y -48.143,Z -63.345,A -90.000,B 90.000,C 0.000} C_DIS
LIN {X 84.510,Y -48.108,Z -63.119,A -90.000,B 90.000,C 0.000} C_DIS
LIN {X 84.505,Y -48.091,Z -62.950,A -90.000,B 90.000,C 0.000} C_DIS
LIN {X 84.505,Y -48.081,Z -62.834,A -90.000,B 90.000,C 0.000} C_DIS
LIN {X 84.512,Y -48.055,Z -62.598,A -90.000,B 90.000,C 0.000} C_DIS
LIN {X 84.519,Y -48.044,Z -62.462,A -90.000,B 90.000,C 0.000} C_DIS
LIN {X 84.582,Y -47.985,Z -61.990,A -90.000,B 90.000,C 0.000} C_DIS
LIN {X 84.631,Y -47.946,Z -61.686,A -90.000,B 90.000,C 0.000} C_DIS
LIN {X 84.645,Y -47.937,Z -61.604,A -90.000,B 90.000,C 0.000} C_DIS
LIN {X 84.664,Y -47.930,Z -61.514,A -90.000,B 90.000,C 0.000} C_DIS
LIN {X 84.677,Y -47.926,Z -61.454,A -90.000,B 90.000,C 0.000} C_DIS
LIN {X 84.869,Y -47.850,Z -60.761,A -90.000,B 90.000,C 0.000} C_DIS
LIN {X 84.895,Y -47.841,Z -60.673,A -90.000,B 90.000,C 0.000} C_DIS
LIN {X 84.960,Y -47.825,Z -60.469,A -90.000,B 90.000,C 0.000} C_DIS
LIN {X 85.104,Y -47.782,Z -60.084,A -90.000,B 90.000,C 0.000} C_DIS
LIN {X 85.140,Y -47.772,Z -59.989,A -90.000,B 90.000,C 0.000} C_DIS
LIN {X 85.197,Y -47.762,Z -59.849,A -90.000,B 90.000,C 0.000} C_DIS
LIN {X 85.362,Y -47.740,Z -59.479,A -90.000,B 90.000,C 0.000} C_DIS
LIN {X 85.580,Y -47.721,Z -59.044,A -90.000,B 90.000,C 0.000} C_DIS
LIN {X 85.690,Y -47.708,Z -58.839,A -90.000,B 90.000,C 0.000} C_DIS
LIN {X 85.734,Y -47.705,Z -58.761,A -90.000,B 90.000,C 0.000} C_DIS
LIN {X 85.802,Y -47.699,Z -58.647,A -90.000,B 90.000,C 0.000} C_DIS
LIN {X 86.026,Y -47.668,Z -58.312,A -90.000,B 90.000,C 0.000} C_DIS
LIN {X 86.173,Y -47.649,Z -58.095,A -90.000,B 90.000,C 0.000} C_DIS
LIN {X 86.649,Y -47.578,Z -57.447,A -90.000,B 90.000,C 0.000} C_DIS
LIN {X 86.783,Y -47.564,Z -57.268,A -90.000,B 90.000,C 0.000} C_DIS
LIN {X 87.022,Y -47.540,Z -56.956,A -90.000,B 90.000,C 0.000} C_DIS
LIN {X 87.196,Y -47.524,Z -56.736,A -90.000,B 90.000,C 0.000} C_DIS
LIN {X 87.444,Y -47.508,Z -56.426,A -90.000,B 90.000,C 0.000} C_DIS
LIN {X 87.583,Y -47.508,Z -56.258,A -90.000,B 90.000,C 0.000} C_DIS
LIN {X 87.775,Y -47.511,Z -56.025,A -90.000,B 90.000,C 0.000} C_DIS
LIN {X 88.095,Y -47.504,Z -55.700,A -90.000,B 90.000,C 0.000} C_DIS
LIN {X 88.792,Y -47.481,Z -55.014,A -90.000,B 90.000,C 0.000} C_DIS
LIN {X 89.756,Y -47.462,Z -54.070,A -90.000,B 90.000,C 0.000} C_DIS
LIN {X 90.041,Y -47.462,Z -53.798,A -90.000,B 90.000,C 0.000} C_DIS
LIN {X 90.121,Y -47.464,Z -53.722,A -90.000,B 90.000,C 0.000} C_DIS
LIN {X 92.269,Y -47.472,Z -51.900,A -90.000,B 90.000,C 0.000} C_DIS
LIN {X 92.524,Y -47.476,Z -51.697,A -90.000,B 90.000,C 0.000} C_DIS
LIN {X 93.247,Y -47.493,Z -51.131,A -90.000,B 90.000,C 0.000} C_DIS
LIN {X 94.259,Y -47.531,Z -50.341,A -90.000,B 90.000,C 0.000} C_DIS
LIN {X 94.680,Y -47.544,Z -50.023,A -90.000,B 90.000,C 0.000} C_DIS
LIN {X 94.821,Y -47.546,Z -49.921,A -90.000,B 90.000,C 0.000} C_DIS
LIN {X 94.938,Y -47.549,Z -49.835,A -90.000,B 90.000,C 0.000} C_DIS
LIN {X 95.404,Y -47.574,Z -49.502,A -90.000,B 90.000,C 0.000} C_DIS
LIN {X 95.991,Y -47.619,Z -49.091,A -90.000,B 90.000,C 0.000} C_DIS
LIN {X 96.721,Y -47.675,Z -48.593,A -90.000,B 90.000,C 0.000} C_DIS
LIN {X 97.146,Y -47.713,Z -48.316,A -90.000,B 90.000,C 0.000} C_DIS
LIN {X 97.562,Y -47.758,Z -48.050,A -90.000,B 90.000,C 0.000} C_DIS
LIN {X 97.763,Y -47.780,Z -47.937,A -90.000,B 90.000,C 0.000} C_DIS
LIN {X 98.196,Y -47.834,Z -47.698,A -90.000,B 90.000,C 0.000} C_DIS
LIN {X 98.498,Y -47.881,Z -47.538,A -90.000,B 90.000,C 0.000} C_DIS
LIN {X 98.635,Y -47.899,Z -47.475,A -90.000,B 90.000,C 0.000} C_DIS
LIN {X 99.186,Y -47.983,Z -47.233,A -90.000,B 90.000,C 0.000} C_DIS
LIN {X 99.305,Y -47.999,Z -47.183,A -90.000,B 90.000,C 0.000} C_DIS
LIN {X 99.417,Y -48.017,Z -47.140,A -90.000,B 90.000,C 0.000} C_DIS
LIN {X 99.590,Y -48.049,Z -47.076,A -90.000,B 90.000,C 0.000} C_DIS
LIN {X 99.778,Y -48.073,Z -47.018,A -90.000,B 90.000,C 0.000} C_DIS
LIN {X 100.067,Y -48.119,Z -46.940,A -90.000,B 90.000,C 0.000} C_DIS
LIN {X 100.235,Y -48.148,Z -46.896,A -90.000,B 90.000,C 0.000} C_DIS
LIN {X 100.449,Y -48.174,Z -46.848,A -90.000,B 90.000,C 0.000} C_DIS
LIN {X 100.543,Y -48.188,Z -46.831,A -90.000,B 90.000,C 0.000} C_DIS
LIN {X 100.851,Y -48.229,Z -46.782,A -90.000,B 90.000,C 0.000} C_DIS
LIN {X 101.006,Y -48.255,Z -46.764,A -90.000,B 90.000,C 0.000} C_DIS
LIN {X 101.089,Y -48.272,Z -46.758,A -90.000,B 90.000,C 0.000} C_DIS
LIN {X 101.429,Y -48.321,Z -46.758,A -90.000,B 90.000,C 0.000} C_DIS
LIN {X 101.555,Y -48.339,Z -46.763,A -90.000,B 90.000,C 0.000} C_DIS
LIN {X 101.693,Y -48.362,Z -46.771,A -90.000,B 90.000,C 0.000} C_DIS
LIN {X 101.817,Y -48.384,Z -46.782,A -90.000,B 90.000,C 0.000} C_DIS
LIN {X 102.100,Y -48.423,Z -46.831,A -90.000,B 90.000,C 0.000} C_DIS
LIN {X 102.252,Y -48.439,Z -46.862,A -90.000,B 90.000,C 0.000} C_DIS
LIN {X 102.435,Y -48.459,Z -46.905,A -90.000,B 90.000,C 0.000} C_DIS
LIN {X 102.576,Y -48.476,Z -46.950,A -90.000,B 90.000,C 0.000} C_DIS
LIN {X 102.696,Y -48.493,Z -46.992,A -90.000,B 90.000,C 0.000} C_DIS
LIN {X 102.722,Y -48.494,Z -47.003,A -90.000,B 90.000,C 0.000} C_DIS
LIN {X 102.881,Y -48.504,Z -47.064,A -90.000,B 90.000,C 0.000} C_DIS
LIN {X 103.000,Y -48.513,Z -47.115,A -90.000,B 90.000,C 0.000} C_DIS
LIN {X 103.104,Y -48.519,Z -47.169,A -90.000,B 90.000,C 0.000} C_DIS
LIN {X 103.328,Y -48.533,Z -47.296,A -90.000,B 90.000,C 0.000} C_DIS
LIN {X 103.470,Y -48.543,Z -47.384,A -90.000,B 90.000,C 0.000} C_DIS
LIN {X 103.616,Y -48.547,Z -47.484,A -90.000,B 90.000,C 0.000} C_DIS
LIN {X 103.728,Y -48.551,Z -47.565,A -90.000,B 90.000,C 0.000} C_DIS
LIN {X 103.754,Y -48.552,Z -47.586,A -90.000,B 90.000,C 0.000} C_DIS
LIN {X 103.863,Y -48.554,Z -47.685,A -90.000,B 90.000,C 0.000} C_DIS
LIN {X 103.980,Y -48.555,Z -47.799,A -90.000,B 90.000,C 0.000} C_DIS
LIN {X 104.099,Y -48.550,Z -47.920,A -90.000,B 90.000,C 0.000} C_DIS
LIN {X 104.176,Y -48.548,Z -48.007,A -90.000,B 90.000,C 0.000} C_DIS
LIN {X 104.370,Y -48.534,Z -48.268,A -90.000,B 90.000,C 0.000} C_DIS
LIN {X 104.467,Y -48.521,Z -48.422,A -90.000,B 90.000,C 0.000} C_DIS
LIN {X 104.525,Y -48.514,Z -48.522,A -90.000,B 90.000,C 0.000} C_DIS
LIN {X 104.646,Y -48.483,Z -48.749,A -90.000,B 90.000,C 0.000} C_DIS
LIN {X 104.693,Y -48.472,Z -48.848,A -90.000,B 90.000,C 0.000} C_DIS
LIN {X 104.737,Y -48.464,Z -48.955,A -90.000,B 90.000,C 0.000} C_DIS
LIN {X 104.799,Y -48.452,Z -49.121,A -90.000,B 90.000,C 0.000} C_DIS
LIN {X 104.858,Y -48.432,Z -49.292,A -90.000,B 90.000,C 0.000} C_DIS
LIN {X 104.903,Y -48.419,Z -49.442,A -90.000,B 90.000,C 0.000} C_DIS
LIN {X 104.984,Y -48.384,Z -49.742,A -90.000,B 90.000,C 0.000} C_DIS
LIN {X 104.995,Y -48.377,Z -49.785,A -90.000,B 90.000,C 0.000} C_DIS
LIN {X 105.017,Y -48.356,Z -49.896,A -90.000,B 90.000,C 0.000} C_DIS
LIN {X 105.072,Y -48.300,Z -50.262,A -90.000,B 90.000,C 0.000} C_DIS
LIN {X 105.086,Y -48.287,Z -50.365,A -90.000,B 90.000,C 0.000} C_DIS
LIN {X 105.094,Y -48.276,Z -50.466,A -90.000,B 90.000,C 0.000} C_DIS
LIN {X 105.110,Y -48.245,Z -50.907,A -90.000,B 90.000,C 0.000} C_DIS
LIN {X 105.104,Y -48.230,Z -51.076,A -90.000,B 90.000,C 0.000} C_DIS
LIN {X 105.091,Y -48.223,Z -51.224,A -90.000,B 90.000,C 0.000} C_DIS
LIN {X 105.074,Y -48.219,Z -51.355,A -90.000,B 90.000,C 0.000} C_DIS
LIN {X 105.031,Y -48.213,Z -51.737,A -90.000,B 90.000,C 0.000} C_DIS
LIN {X 104.988,Y -48.204,Z -52.095,A -90.000,B 90.000,C 0.000} C_DIS
LIN {X 104.962,Y -48.202,Z -52.268,A -90.000,B 90.000,C 0.000} C_DIS
LIN {X 104.941,Y -48.193,Z -52.475,A -90.000,B 90.000,C 0.000} C_DIS
LIN {X 104.930,Y -48.191,Z -52.571,A -90.000,B 90.000,C 0.000} C_DIS
LIN {X 104.913,Y -48.186,Z -52.713,A -90.000,B 90.000,C 0.000} C_DIS
LIN {X 104.883,Y -48.174,Z -52.907,A -90.000,B 90.000,C 0.000} C_DIS
LIN {X 104.860,Y -48.172,Z -53.015,A -90.000,B 90.000,C 0.000} C_DIS
LIN {X 104.774,Y -48.174,Z -53.402,A -90.000,B 90.000,C 0.000} C_DIS
LIN {X 104.720,Y -48.168,Z -53.693,A -90.000,B 90.000,C 0.000} C_DIS
LIN {X 104.680,Y -48.170,Z -53.938,A -90.000,B 90.000,C 0.000} C_DIS
LIN {X 104.592,Y -48.181,Z -54.411,A -90.000,B 90.000,C 0.000} C_DIS
LIN {X 104.482,Y -48.201,Z -54.912,A -90.000,B 90.000,C 0.000} C_DIS
LIN {X 104.439,Y -48.211,Z -55.080,A -90.000,B 90.000,C 0.000} C_DIS
LIN {X 104.321,Y -48.246,Z -55.471,A -90.000,B 90.000,C 0.000} C_DIS
LIN {X 104.299,Y -48.250,Z -55.540,A -90.000,B 90.000,C 0.000} C_DIS
LIN {X 104.226,Y -48.254,Z -55.804,A -90.000,B 90.000,C 0.000} C_DIS
LIN {X 104.014,Y -48.271,Z -56.456,A -90.000,B 90.000,C 0.000} C_DIS
LIN {X 103.662,Y -48.271,Z -57.685,A -90.000,B 90.000,C 0.000} C_DIS
LIN {X 103.614,Y -48.275,Z -57.827,A -90.000,B 90.000,C 0.000} C_DIS
LIN {X 103.491,Y -48.290,Z -58.160,A -90.000,B 90.000,C 0.000} C_DIS
LIN {X 102.839,Y -48.301,Z -59.725,A -90.000,B 90.000,C 0.000} C_DIS
LIN {X 102.495,Y -48.302,Z -60.568,A -90.000,B 90.000,C 0.000} C_DIS
LIN {X 102.398,Y -48.309,Z -60.776,A -90.000,B 90.000,C 0.000} C_DIS
LIN {X 101.643,Y -48.334,Z -62.125,A -90.000,B 90.000,C 0.000} C_DIS
LIN {X 101.169,Y -48.344,Z -62.963,A -90.000,B 90.000,C 0.000} C_DIS
LIN {X 101.169,Y -60.000,Z -62.963,A -90.000,B 90.000,C 0.000} C_DIS
LIN {X 102.376,Y -60.000,Z -45.186,A -90.000,B 90.000,C 0.000} C_DIS
LIN {X 102.376,Y -47.308,Z -45.186,A -90.000,B 90.000,C 0.000} C_DIS
LIN {X 102.534,Y -47.353,Z -45.198,A -90.000,B 90.000,C 0.000} C_DIS
LIN {X 102.804,Y -47.421,Z -45.230,A -90.000,B 90.000,C 0.000} C_DIS
LIN {X 102.937,Y -47.447,Z -45.255,A -90.000,B 90.000,C 0.000} C_DIS
LIN {X 103.069,Y -47.476,Z -45.284,A -90.000,B 90.000,C 0.000} C_DIS
LIN {X 103.231,Y -47.512,Z -45.325,A -90.000,B 90.000,C 0.000} C_DIS
LIN {X 103.431,Y -47.559,Z -45.383,A -90.000,B 90.000,C 0.000} C_DIS
LIN {X 103.716,Y -47.604,Z -45.483,A -90.000,B 90.000,C 0.000} C_DIS
LIN {X 103.787,Y -47.613,Z -45.512,A -90.000,B 90.000,C 0.000} C_DIS
LIN {X 103.968,Y -47.640,Z -45.594,A -90.000,B 90.000,C 0.000} C_DIS
LIN {X 104.227,Y -47.675,Z -45.728,A -90.000,B 90.000,C 0.000} C_DIS
LIN {X 104.329,Y -47.683,Z -45.788,A -90.000,B 90.000,C 0.000} C_DIS
LIN {X 104.524,Y -47.699,Z -45.908,A -90.000,B 90.000,C 0.000} C_DIS
LIN {X 104.710,Y -47.708,Z -46.034,A -90.000,B 90.000,C 0.000} C_DIS
LIN {X 104.889,Y -47.717,Z -46.167,A -90.000,B 90.000,C 0.000} C_DIS
LIN {X 104.937,Y -47.720,Z -46.205,A -90.000,B 90.000,C 0.000} C_DIS
LIN {X 105.135,Y -47.724,Z -46.384,A -90.000,B 90.000,C 0.000} C_DIS
LIN {X 105.172,Y -47.725,Z -46.420,A -90.000,B 90.000,C 0.000} C_DIS
LIN {X 105.395,Y -47.714,Z -46.646,A -90.000,B 90.000,C 0.000} C_DIS
LIN {X 105.523,Y -47.699,Z -46.796,A -90.000,B 90.000,C 0.000} C_DIS
LIN {X 105.593,Y -47.692,Z -46.884,A -90.000,B 90.000,C 0.000} C_DIS
LIN {X 105.776,Y -47.656,Z -47.149,A -90.000,B 90.000,C 0.000} C_DIS
LIN {X 105.847,Y -47.637,Z -47.260,A -90.000,B 90.000,C 0.000} C_DIS
LIN {X 105.961,Y -47.607,Z -47.455,A -90.000,B 90.000,C 0.000} C_DIS
LIN {X 106.110,Y -47.563,Z -47.741,A -90.000,B 90.000,C 0.000} C_DIS
LIN {X 106.176,Y -47.542,Z -47.871,A -90.000,B 90.000,C 0.000} C_DIS
LIN {X 106.212,Y -47.531,Z -47.947,A -90.000,B 90.000,C 0.000} C_DIS
LIN {X 106.280,Y -47.495,Z -48.122,A -90.000,B 90.000,C 0.000} C_DIS
LIN {X 106.311,Y -47.479,Z -48.212,A -90.000,B 90.000,C 0.000} C_DIS
LIN {X 106.416,Y -47.414,Z -48.556,A -90.000,B 90.000,C 0.000} C_DIS
LIN {X 106.459,Y -47.376,Z -48.725,A -90.000,B 90.000,C 0.000} C_DIS
LIN {X 106.534,Y -47.308,Z -49.066,A -90.000,B 90.000,C 0.000} C_DIS
LIN {X 106.534,Y -60.000,Z -49.066,A -90.000,B 90.000,C 0.000} C_DIS
LIN {X 102.308,Y -60.000,Z -64.379,A -90.000,B 90.000,C 0.000} C_DIS
LIN {X 102.308,Y -47.308,Z -64.379,A -90.000,B 90.000,C 0.000} C_DIS
LIN {X 102.275,Y -47.311,Z -64.423,A -90.000,B 90.000,C 0.000} C_DIS
LIN {X 102.172,Y -47.315,Z -64.576,A -90.000,B 90.000,C 0.000} C_DIS
LIN {X 101.892,Y -47.336,Z -64.964,A -90.000,B 90.000,C 0.000} C_DIS
LIN {X 101.812,Y -47.343,Z -65.068,A -90.000,B 90.000,C 0.000} C_DIS
LIN {X 100.979,Y -47.434,Z -66.132,A -90.000,B 90.000,C 0.000} C_DIS
LIN {X 100.739,Y -47.439,Z -66.420,A -90.000,B 90.000,C 0.000} C_DIS
LIN {X 100.453,Y -47.433,Z -66.753,A -90.000,B 90.000,C 0.000} C_DIS
LIN {X 100.131,Y -47.433,Z -67.109,A -90.000,B 90.000,C 0.000} C_DIS
LIN {X 100.068,Y -47.434,Z -67.175,A -90.000,B 90.000,C 0.000} C_DIS
LIN {X 99.884,Y -47.443,Z -67.354,A -90.000,B 90.000,C 0.000} C_DIS
LIN {X 99.772,Y -47.450,Z -67.460,A -90.000,B 90.000,C 0.000} C_DIS
LIN {X 99.467,Y -47.473,Z -67.721,A -90.000,B 90.000,C 0.000} C_DIS
LIN {X 99.363,Y -47.482,Z -67.805,A -90.000,B 90.000,C 0.000} C_DIS
LIN {X 98.802,Y -47.539,Z -68.238,A -90.000,B 90.000,C 0.000} C_DIS
LIN {X 98.537,Y -47.549,Z -68.430,A -90.000,B 90.000,C 0.000} C_DIS
LIN {X 98.191,Y -47.554,Z -68.677,A -90.000,B 90.000,C 0.000} C_DIS
LIN {X 98.086,Y -47.558,Z -68.746,A -90.000,B 90.000,C 0.000} C_DIS
LIN {X 97.749,Y -47.577,Z -68.955,A -90.000,B 90.000,C 0.000} C_DIS
LIN {X 97.596,Y -47.587,Z -69.046,A -90.000,B 90.000,C 0.000} C_DIS
LIN {X 97.288,Y -47.612,Z -69.220,A -90.000,B 90.000,C 0.000} C_DIS
LIN {X 96.778,Y -47.643,Z -69.502,A -90.000,B 90.000,C 0.000} C_DIS
LIN {X 96.504,Y -47.649,Z -69.649,A -90.000,B 90.000,C 0.000} C_DIS
LIN {X 96.435,Y -47.647,Z -69.686,A -90.000,B 90.000,C 0.000} C_DIS
LIN {X 96.297,Y -47.647,Z -69.754,A -90.000,B 90.000,C 0.000} C_DIS
LIN {X 96.039,Y -47.652,Z -69.869,A -90.000,B 90.000,C 0.000} C_DIS
LIN {X 95.552,Y -47.669,Z -70.064,A -90.000,B 90.000,C 0.000} C_DIS
LIN {X 95.380,Y -47.678,Z -70.122,A -90.000,B 90.000,C 0.000} C_DIS
LIN {X 95.257,Y -47.682,Z -70.161,A -90.000,B 90.000,C 0.000} C_DIS
LIN {X 95.190,Y -47.685,Z -70.181,A -90.000,B 90.000,C 0.000} C_DIS
LIN {X 95.057,Y -47.690,Z -70.216,A -90.000,B 90.000,C 0.000} C_DIS
LIN {X 94.852,Y -47.691,Z -70.267,A -90.000,B 90.000,C 0.000} C_DIS
LIN {X 94.166,Y -47.708,Z -70.442,A -90.000,B 90.000,C 0.000} C_DIS
LIN {X 93.993,Y -47.714,Z -70.482,A -90.000,B 90.000,C 0.000} C_DIS
LIN {X 93.689,Y -47.714,Z -70.547,A -90.000,B 90.000,C 0.000} C_DIS
LIN {X 93.541,Y -47.711,Z -70.568,A -90.000,B 90.000,C 0.000} C_DIS
LIN {X 93.340,Y -47.710,Z -70.589,A -90.000,B 90.000,C 0.000} C_DIS
LIN {X 92.953,Y -47.714,Z -70.614,A -90.000,B 90.000,C 0.000} C_DIS
LIN {X 92.598,Y -47.728,Z -70.637,A -90.000,B 90.000,C 0.000} C_DIS
LIN {X 92.410,Y -47.730,Z -70.645,A -90.000,B 90.000,C 0.000} C_DIS
LIN {X 92.298,Y -47.732,Z -70.647,A -90.000,B 90.000,C 0.000} C_DIS
LIN {X 91.646,Y -47.721,Z -70.630,A -90.000,B 90.000,C 0.000} C_DIS
LIN {X 91.353,Y -47.719,Z -70.617,A -90.000,B 90.000,C 0.000} C_DIS
LIN {X 91.107,Y -47.712,Z -70.625,A -90.000,B 90.000,C 0.000} C_DIS
LIN {X 90.925,Y -47.700,Z -70.625,A -90.000,B 90.000,C 0.000} C_DIS
LIN {X 90.761,Y -47.690,Z -70.618,A -90.000,B 90.000,C 0.000} C_DIS
LIN {X 90.519,Y -47.680,Z -70.596,A -90.000,B 90.000,C 0.000} C_DIS
LIN {X 90.176,Y -47.671,Z -70.558,A -90.000,B 90.000,C 0.000} C_DIS
LIN {X 89.937,Y -47.668,Z -70.520,A -90.000,B 90.000,C 0.000} C_DIS
LIN {X 89.754,Y -47.663,Z -70.485,A -90.000,B 90.000,C 0.000} C_DIS
LIN {X 89.614,Y -47.660,Z -70.456,A -90.000,B 90.000,C 0.000} C_DIS
LIN {X 89.283,Y -47.637,Z -70.378,A -90.000,B 90.000,C 0.000} C_DIS
LIN {X 88.991,Y -47.616,Z -70.302,A -90.000,B 90.000,C 0.000} C_DIS
LIN {X 88.700,Y -47.590,Z -70.225,A -90.000,B 90.000,C 0.000} C_DIS
LIN {X 88.551,Y -47.583,Z -70.188,A -90.000,B 90.000,C 0.000} C_DIS
LIN {X 88.136,Y -47.571,Z -70.074,A -90.000,B 90.000,C 0.000} C_DIS
LIN {X 87.983,Y -47.564,Z -70.023,A -90.000,B 90.000,C 0.000} C_DIS
LIN {X 87.831,Y -47.559,Z -69.967,A -90.000,B 90.000,C 0.000} C_DIS
LIN {X 87.699,Y -47.548,Z -69.910,A -90.000,B 90.000,C 0.000} C_DIS
LIN {X 87.519,Y -47.535,Z -69.826,A -90.000,B 90.000,C 0.000} C_DIS
LIN {X 87.241,Y -47.514,Z -69.690,A -90.000,B 90.000,C 0.000} C_DIS
LIN {X 87.158,Y -47.509,Z -69.647,A -90.000,B 90.000,C 0.000} C_DIS
LIN {X 86.832,Y -47.509,Z -69.486,A -90.000,B 90.000,C 0.000} C_DIS
LIN {X 86.540,Y -47.499,Z -69.321,A -90.000,B 90.000,C 0.000} C_DIS
LIN {X 86.311,Y -47.475,Z -69.182,A -90.000,B 90.000,C 0.000} C_DIS
LIN {X 86.206,Y -47.461,Z -69.116,A -90.000,B 90.000,C 0.000} C_DIS
LIN {X 86.056,Y -47.443,Z -69.016,A -90.000,B 90.000,C 0.000} C_DIS
LIN {X 85.990,Y -47.437,Z -68.969,A -90.000,B 90.000,C 0.000} C_DIS
LIN {X 85.746,Y -47.428,Z -68.808,A -90.000,B 90.000,C 0.000} C_DIS
LIN {X 85.629,Y -47.425,Z -68.724,A -90.000,B 90.000,C 0.000} C_DIS
LIN {X 85.520,Y -47.423,Z -68.643,A -90.000,B 90.000,C 0.000} C_DIS
LIN {X 85.355,Y -47.413,Z -68.499,A -90.000,B 90.000,C 0.000} C_DIS
LIN {X 85.259,Y -47.408,Z -68.411,A -90.000,B 90.000,C 0.000} C_DIS
LIN {X 85.127,Y -47.389,Z -68.280,A -90.000,B 90.000,C 0.000} C_DIS
LIN {X 85.008,Y -47.373,Z -68.156,A -90.000,B 90.000,C 0.000} C_DIS
LIN {X 84.898,Y -47.356,Z -68.031,A -90.000,B 90.000,C 0.000} C_DIS
LIN {X 84.833,Y -47.347,Z -67.953,A -90.000,B 90.000,C 0.000} C_DIS
LIN {X 84.665,Y -47.335,Z -67.772,A -90.000,B 90.000,C 0.000} C_DIS
LIN {X 84.466,Y -47.315,Z -67.552,A -90.000,B 90.000,C 0.000} C_DIS
LIN {X 84.430,Y -47.308,Z -67.510,A -90.000,B 90.000,C 0.000} C_DIS
LIN {X 84.345,Y -47.308,Z -67.368,A -90.000,B 90.000,C 0.000} C_DIS
LIN {X 84.168,Y -47.308,Z -67.033,A -90.000,B 90.000,C 0.000} C_DIS
LIN {X 84.037,Y -47.308,Z -66.677,A -90.000,B 90.000,C 0.000} C_DIS
LIN {X 83.862,Y -47.308,Z -66.078,A -90.000,B 90.000,C 0.000} C_DIS
LIN {X 83.738,Y -47.308,Z -65.613,A -90.000,B 90.000,C 0.000} C_DIS
LIN {X 83.702,Y -47.308,Z -65.454,A -90.000,B 90.000,C 0.000} C_DIS
LIN {X 83.669,Y -47.308,Z -65.226,A -90.000,B 90.000,C 0.000} C_DIS
LIN {X 83.643,Y -47.308,Z -64.957,A -90.000,B 90.000,C 0.000} C_DIS
LIN {X 83.634,Y -47.308,Z -64.554,A -90.000,B 90.000,C 0.000} C_DIS
LIN {X 83.678,Y -47.308,Z -63.917,A -90.000,B 90.000,C 0.000} C_DIS
LIN {X 83.733,Y -47.308,Z -63.498,A -90.000,B 90.000,C 0.000} C_DIS
LIN {X 83.793,Y -47.308,Z -63.140,A -90.000,B 90.000,C 0.000} C_DIS
LIN {X 83.971,Y -47.308,Z -62.172,A -90.000,B 90.000,C 0.000} C_DIS
LIN {X 84.073,Y -47.308,Z -61.772,A -90.000,B 90.000,C 0.000} C_DIS
LIN {X 84.080,Y -47.308,Z -61.745,A -90.000,B 90.000,C 0.000} C_DIS
LIN {X 84.110,Y -47.308,Z -61.632,A -90.000,B 90.000,C 0.000} C_DIS
LIN {X 84.139,Y -47.308,Z -61.550,A -90.000,B 90.000,C 0.000} C_DIS
LIN {X 84.266,Y -47.308,Z -61.217,A -90.000,B 90.000,C 0.000} C_DIS
LIN {X 84.531,Y -47.308,Z -60.629,A -90.000,B 90.000,C 0.000} C_DIS
LIN {X 84.730,Y -47.308,Z -60.220,A -90.000,B 90.000,C 0.000} C_DIS
LIN {X 85.098,Y -47.308,Z -59.521,A -90.000,B 90.000,C 0.000} C_DIS
LIN {X 85.330,Y -47.308,Z -59.115,A -90.000,B 90.000,C 0.000} C_DIS
LIN {X 85.560,Y -47.308,Z -58.729,A -90.000,B 90.000,C 0.000} C_DIS
LIN {X 85.710,Y -47.308,Z -58.494,A -90.000,B 90.000,C 0.000} C_DIS
LIN {X 85.824,Y -47.308,Z -58.337,A -90.000,B 90.000,C 0.000} C_DIS
LIN {X 86.162,Y -47.308,Z -57.907,A -90.000,B 90.000,C 0.000} C_DIS
LIN {X 86.460,Y -47.308,Z -57.535,A -90.000,B 90.000,C 0.000} C_DIS
LIN {X 86.826,Y -47.308,Z -57.088,A -90.000,B 90.000,C 0.000} C_DIS
LIN {X 87.635,Y -47.308,Z -56.112,A -90.000,B 90.000,C 0.000} C_DIS
LIN {X 87.779,Y -47.308,Z -55.943,A -90.000,B 90.000,C 0.000} C_DIS
LIN {X 87.960,Y -47.308,Z -55.760,A -90.000,B 90.000,C 0.000} C_DIS
LIN {X 89.407,Y -47.308,Z -54.353,A -90.000,B 90.000,C 0.000} C_DIS
LIN {X 90.128,Y -47.308,Z -53.670,A -90.000,B 90.000,C 0.000} C_DIS
LIN {X 92.282,Y -47.308,Z -51.834,A -90.000,B 90.000,C 0.000} C_DIS
LIN {X 94.575,Y -47.308,Z -50.017,A -90.000,B 90.000,C 0.000} C_DIS
LIN {X 95.229,Y -47.308,Z -49.505,A -90.000,B 90.000,C 0.000} C_DIS
LIN {X 96.607,Y -47.308,Z -48.485,A -90.000,B 90.000,C 0.000} C_DIS
LIN {X 96.675,Y -47.308,Z -48.433,A -90.000,B 90.000,C 0.000} C_DIS
LIN {X 97.125,Y -47.308,Z -48.096,A -90.000,B 90.000,C 0.000} C_DIS
LIN {X 97.502,Y -47.308,Z -47.825,A -90.000,B 90.000,C 0.000} C_DIS
LIN {X 98.576,Y -47.308,Z -47.067,A -90.000,B 90.000,C 0.000} C_DIS
LIN {X 98.992,Y -47.308,Z -46.801,A -90.000,B 90.000,C 0.000} C_DIS
LIN {X 99.581,Y -47.308,Z -46.434,A -90.000,B 90.000,C 0.000} C_DIS
LIN {X 99.962,Y -47.308,Z -46.213,A -90.000,B 90.000,C 0.000} C_DIS
LIN {X 100.872,Y -47.308,Z -45.732,A -90.000,B 90.000,C 0.000} C_DIS
LIN {X 101.021,Y -47.308,Z -45.666,A -90.000,B 90.000,C 0.000} C_DIS
LIN {X 101.612,Y -47.308,Z -45.429,A -90.000,B 90.000,C 0.000} C_DIS
LIN {X 101.990,Y -47.308,Z -45.290,A -90.000,B 90.000,C 0.000} C_DIS
LIN {X 102.599,Y -47.308,Z -45.126,A -90.000,B 90.000,C 0.000} C_DIS
LIN {X 102.970,Y -47.308,Z -45.047,A -90.000,B 90.000,C 0.000} C_DIS
LIN {X 103.446,Y -47.308,Z -44.999,A -90.000,B 90.000,C 0.000} C_DIS
LIN {X 103.797,Y -47.308,Z -44.976,A -90.000,B 90.000,C 0.000} C_DIS
LIN {X 104.149,Y -47.308,Z -45.003,A -90.000,B 90.000,C 0.000} C_DIS
LIN {X 104.492,Y -47.308,Z -45.080,A -90.000,B 90.000,C 0.000} C_DIS
LIN {X 104.745,Y -47.308,Z -45.151,A -90.000,B 90.000,C 0.000} C_DIS
LIN {X 105.040,Y -47.308,Z -45.274,A -90.000,B 90.000,C 0.000} C_DIS
LIN {X 105.173,Y -47.308,Z -45.352,A -90.000,B 90.000,C 0.000} C_DIS
LIN {X 105.240,Y -47.308,Z -45.387,A -90.000,B 90.000,C 0.000} C_DIS
LIN {X 105.512,Y -47.308,Z -45.555,A -90.000,B 90.000,C 0.000} C_DIS
LIN {X 105.754,Y -47.308,Z -45.763,A -90.000,B 90.000,C 0.000} C_DIS
LIN {X 105.960,Y -47.308,Z -46.007,A -90.000,B 90.000,C 0.000} C_DIS
LIN {X 106.127,Y -47.308,Z -46.279,A -90.000,B 90.000,C 0.000} C_DIS
LIN {X 106.236,Y -47.308,Z -46.542,A -90.000,B 90.000,C 0.000} C_DIS
LIN {X 106.357,Y -47.308,Z -46.867,A -90.000,B 90.000,C 0.000} C_DIS
LIN {X 106.449,Y -47.308,Z -47.222,A -90.000,B 90.000,C 0.000} C_DIS
LIN {X 106.528,Y -47.308,Z -47.581,A -90.000,B 90.000,C 0.000} C_DIS
LIN {X 106.556,Y -47.308,Z -47.991,A -90.000,B 90.000,C 0.000} C_DIS
LIN {X 106.566,Y -47.308,Z -48.383,A -90.000,B 90.000,C 0.000} C_DIS
LIN {X 106.556,Y -47.308,Z -48.616,A -90.000,B 90.000,C 0.000} C_DIS
LIN {X 106.540,Y -47.308,Z -48.901,A -90.000,B 90.000,C 0.000} C_DIS
LIN {X 106.526,Y -47.308,Z -49.245,A -90.000,B 90.000,C 0.000} C_DIS
LIN {X 106.486,Y -47.308,Z -49.561,A -90.000,B 90.000,C 0.000} C_DIS
LIN {X 106.431,Y -47.308,Z -50.034,A -90.000,B 90.000,C 0.000} C_DIS
LIN {X 106.345,Y -47.308,Z -50.736,A -90.000,B 90.000,C 0.000} C_DIS
LIN {X 106.303,Y -47.308,Z -51.007,A -90.000,B 90.000,C 0.000} C_DIS
LIN {X 106.238,Y -47.308,Z -51.559,A -90.000,B 90.000,C 0.000} C_DIS
LIN {X 106.233,Y -47.308,Z -51.917,A -90.000,B 90.000,C 0.000} C_DIS
LIN {X 106.241,Y -47.308,Z -52.056,A -90.000,B 90.000,C 0.000} C_DIS
LIN {X 106.250,Y -47.308,Z -52.632,A -90.000,B 90.000,C 0.000} C_DIS
LIN {X 106.249,Y -47.308,Z -52.697,A -90.000,B 90.000,C 0.000} C_DIS
LIN {X 106.255,Y -47.308,Z -52.839,A -90.000,B 90.000,C 0.000} C_DIS
LIN {X 106.231,Y -47.308,Z -53.539,A -90.000,B 90.000,C 0.000} C_DIS
LIN {X 106.170,Y -47.308,Z -54.173,A -90.000,B 90.000,C 0.000} C_DIS
LIN {X 105.997,Y -47.308,Z -55.071,A -90.000,B 90.000,C 0.000} C_DIS
LIN {X 105.779,Y -47.308,Z -55.972,A -90.000,B 90.000,C 0.000} C_DIS
LIN {X 105.561,Y -47.308,Z -56.806,A -90.000,B 90.000,C 0.000} C_DIS
LIN {X 105.376,Y -47.308,Z -57.380,A -90.000,B 90.000,C 0.000} C_DIS
LIN {X 104.822,Y -47.308,Z -59.028,A -90.000,B 90.000,C 0.000} C_DIS
LIN {X 104.228,Y -47.308,Z -60.481,A -90.000,B 90.000,C 0.000} C_DIS
LIN {X 103.967,Y -47.308,Z -61.110,A -90.000,B 90.000,C 0.000} C_DIS
LIN {X 103.902,Y -47.308,Z -61.270,A -90.000,B 90.000,C 0.000} C_DIS
LIN {X 103.749,Y -47.308,Z -61.617,A -90.000,B 90.000,C 0.000} C_DIS
LIN {X 102.935,Y -47.308,Z -63.235,A -90.000,B 90.000,C 0.000} C_DIS
LIN {X 102.671,Y -47.308,Z -63.778,A -90.000,B 90.000,C 0.000} C_DIS
LIN {X 102.495,Y -47.308,Z -64.082,A -90.000,B 90.000,C 0.000} C_DIS
LIN {X 101.520,Y -47.308,Z -65.630,A -90.000,B 90.000,C 0.000} C_DIS
LIN {X 101.161,Y -47.308,Z -66.223,A -90.000,B 90.000,C 0.000} C_DIS
LIN {X 100.944,Y -47.308,Z -66.499,A -90.000,B 90.000,C 0.000} C_DIS
LIN {X 100.372,Y -47.308,Z -67.191,A -90.000,B 90.000,C 0.000} C_DIS
LIN {X 99.214,Y -47.308,Z -68.471,A -90.000,B 90.000,C 0.000} C_DIS
LIN {X 98.954,Y -47.308,Z -68.684,A -90.000,B 90.000,C 0.000} C_DIS
LIN {X 96.862,Y -47.308,Z -70.280,A -90.000,B 90.000,C 0.000} C_DIS
LIN {X 96.619,Y -47.308,Z -70.421,A -90.000,B 90.000,C 0.000} C_DIS
LIN {X 96.348,Y -47.308,Z -70.570,A -90.000,B 90.000,C 0.000} C_DIS
LIN {X 95.352,Y -47.308,Z -71.046,A -90.000,B 90.000,C 0.000} C_DIS
LIN {X 95.054,Y -47.308,Z -71.162,A -90.000,B 90.000,C 0.000} C_DIS
LIN {X 94.185,Y -47.308,Z -71.388,A -90.000,B 90.000,C 0.000} C_DIS
LIN {X 93.947,Y -47.308,Z -71.463,A -90.000,B 90.000,C 0.000} C_DIS
LIN {X 93.635,Y -47.308,Z -71.531,A -90.000,B 90.000,C 0.000} C_DIS
LIN {X 93.524,Y -47.308,Z -71.542,A -90.000,B 90.000,C 0.000} C_DIS
LIN {X 93.462,Y -47.308,Z -71.551,A -90.000,B 90.000,C 0.000} C_DIS
LIN {X 93.417,Y -47.308,Z -71.557,A -90.000,B 90.000,C 0.000} C_DIS
LIN {X 92.401,Y -47.308,Z -71.682,A -90.000,B 90.000,C 0.000} C_DIS
LIN {X 92.120,Y -47.308,Z -71.678,A -90.000,B 90.000,C 0.000} C_DIS
LIN {X 91.637,Y -47.308,Z -71.638,A -90.000,B 90.000,C 0.000} C_DIS
LIN {X 91.089,Y -47.308,Z -71.618,A -90.000,B 90.000,C 0.000} C_DIS
LIN {X 90.907,Y -47.308,Z -71.588,A -90.000,B 90.000,C 0.000} C_DIS
LIN {X 90.413,Y -47.308,Z -71.464,A -90.000,B 90.000,C 0.000} C_DIS
LIN {X 89.907,Y -47.308,Z -71.372,A -90.000,B 90.000,C 0.000} C_DIS
LIN {X 89.598,Y -47.308,Z -71.292,A -90.000,B 90.000,C 0.000} C_DIS
LIN {X 88.937,Y -47.308,Z -71.029,A -90.000,B 90.000,C 0.000} C_DIS
LIN {X 88.644,Y -47.308,Z -70.901,A -90.000,B 90.000,C 0.000} C_DIS
LIN {X 88.034,Y -47.308,Z -70.598,A -90.000,B 90.000,C 0.000} C_DIS
LIN {X 87.865,Y -47.308,Z -70.541,A -90.000,B 90.000,C 0.000} C_DIS
LIN {X 87.572,Y -47.308,Z -70.413,A -90.000,B 90.000,C 0.000} C_DIS
LIN {X 87.315,Y -47.308,Z -70.250,A -90.000,B 90.000,C 0.000} C_DIS
LIN {X 86.759,Y -47.308,Z -69.874,A -90.000,B 90.000,C 0.000} C_DIS
LIN {X 86.640,Y -47.308,Z -69.815,A -90.000,B 90.000,C 0.000} C_DIS
LIN {X 86.370,Y -47.308,Z -69.644,A -90.000,B 90.000,C 0.000} C_DIS
LIN {X 86.171,Y -47.308,Z -69.473,A -90.000,B 90.000,C 0.000} C_DIS
LIN {X 85.783,Y -47.308,Z -69.098,A -90.000,B 90.000,C 0.000} C_DIS
LIN {X 85.694,Y -47.308,Z -69.033,A -90.000,B 90.000,C 0.000} C_DIS
LIN {X 85.416,Y -47.308,Z -68.818,A -90.000,B 90.000,C 0.000} C_DIS
LIN {X 85.172,Y -47.308,Z -68.566,A -90.000,B 90.000,C 0.000} C_DIS
LIN {X 84.966,Y -47.308,Z -68.281,A -90.000,B 90.000,C 0.000} C_DIS
LIN {X 84.784,Y -47.308,Z -67.989,A -90.000,B 90.000,C 0.000} C_DIS
LIN {X 84.667,Y -47.308,Z -67.846,A -90.000,B 90.000,C 0.000} C_DIS
LIN {X 84.461,Y -47.308,Z -67.561,A -90.000,B 90.000,C 0.000} C_DIS
LIN {X 84.430,Y -47.308,Z -67.510,A -90.000,B 90.000,C 0.000} C_DIS
LIN {X 84.338,Y -47.315,Z -67.358,A -90.000,B 90.000,C 0.000} C_DIS
LIN {X 84.252,Y -47.313,Z -67.203,A -90.000,B 90.000,C 0.000} C_DIS
LIN {X 84.165,Y -47.306,Z -67.048,A -90.000,B 90.000,C 0.000} C_DIS
LIN {X 84.009,Y -47.289,Z -66.685,A -90.000,B 90.000,C 0.000} C_DIS
LIN {X 83.903,Y -47.271,Z -66.398,A -90.000,B 90.000,C 0.000} C_DIS
LIN {X 83.717,Y -47.236,Z -65.912,A -90.000,B 90.000,C 0.000} C_DIS
LIN {X 83.625,Y -47.212,Z -65.670,A -90.000,B 90.000,C 0.000} C_DIS
LIN {X 83.582,Y -47.199,Z -65.549,A -90.000,B 90.000,C 0.000} C_DIS
LIN {X 83.515,Y -47.174,Z -65.305,A -90.000,B 90.000,C 0.000} C_DIS
LIN {X 83.460,Y -47.144,Z -65.060,A -90.000,B 90.000,C 0.000} C_DIS
LIN {X 83.439,Y -47.128,Z -64.938,A -90.000,B 90.000,C 0.000} C_DIS
LIN {X 83.399,Y -47.087,Z -64.694,A -90.000,B 90.000,C 0.000} C_DIS
LIN {X 83.365,Y -47.015,Z -64.292,A -90.000,B 90.000,C 0.000} C_DIS
LIN {X 83.352,Y -46.978,Z -64.132,A -90.000,B 90.000,C 0.000} C_DIS
LIN {X 83.345,Y -46.941,Z -63.973,A -90.000,B 90.000,C 0.000} C_DIS
LIN {X 83.336,Y -46.885,Z -63.736,A -90.000,B 90.000,C 0.000} C_DIS
LIN {X 83.329,Y -46.793,Z -63.343,A -90.000,B 90.000,C 0.000} C_DIS
LIN {X 83.334,Y -46.719,Z -63.032,A -90.000,B 90.000,C 0.000} C_DIS
LIN {X 83.338,Y -46.683,Z -62.877,A -90.000,B 90.000,C 0.000} C_DIS
LIN {X 83.348,Y -46.647,Z -62.724,A -90.000,B 90.000,C 0.000} C_DIS
LIN {X 83.358,Y -46.611,Z -62.571,A -90.000,B 90.000,C 0.000} C_DIS
LIN {X 83.376,Y -46.575,Z -62.420,A -90.000,B 90.000,C 0.000} C_DIS
LIN {X 83.404,Y -46.521,Z -62.194,A -90.000,B 90.000,C 0.000} C_DIS
LIN {X 83.433,Y -46.486,Z -62.047,A -90.000,B 90.000,C 0.000} C_DIS
LIN {X 83.501,Y -46.415,Z -61.756,A -90.000,B 90.000,C 0.000} C_DIS
LIN {X 83.581,Y -46.345,Z -61.468,A -90.000,B 90.000,C 0.000} C_DIS
LIN {X 83.674,Y -46.274,Z -61.184,A -90.000,B 90.000,C 0.000} C_DIS
LIN {X 83.806,Y -46.186,Z -60.833,A -90.000,B 90.000,C 0.000} C_DIS
LIN {X 83.981,Y -46.079,Z -60.414,A -90.000,B 90.000,C 0.000} C_DIS
LIN {X 84.082,Y -46.025,Z -60.209,A -90.000,B 90.000,C 0.000} C_DIS
LIN {X 84.234,Y -45.953,Z -59.942,A -90.000,B 90.000,C 0.000} C_DIS
LIN {X 84.442,Y -45.861,Z -59.613,A -90.000,B 90.000,C 0.000} C_DIS
LIN {X 84.617,Y -45.786,Z -59.349,A -90.000,B 90.000,C 0.000} C_DIS
LIN {X 85.059,Y -45.603,Z -58.710,A -90.000,B 90.000,C 0.000} C_DIS
LIN {X 85.399,Y -45.473,Z -58.273,A -90.000,B 90.000,C 0.000} C_DIS
LIN {X 85.618,Y -45.344,Z -57.999,A -90.000,B 90.000,C 0.000} C_DIS
LIN {X 85.732,Y -45.343,Z -57.856,A -90.000,B 90.000,C 0.000} C_DIS
LIN {X 86.060,Y -45.337,Z -57.493,A -90.000,B 90.000,C 0.000} C_DIS
LIN {X 86.623,Y -45.327,Z -56.906,A -90.000,B 90.000,C 0.000} C_DIS
LIN {X 87.736,Y -45.316,Z -55.746,A -90.000,B 90.000,C 0.000} C_DIS
LIN {X 87.806,Y -45.316,Z -55.675,A -90.000,B 90.000,C 0.000} C_DIS
LIN {X 89.812,Y -45.311,Z -53.839,A -90.000,B 90.000,C 0.000} C_DIS
LIN {X 90.146,Y -45.310,Z -53.537,A -90.000,B 90.000,C 0.000} C_DIS
LIN {X 92.378,Y -45.311,Z -51.626,A -90.000,B 90.000,C 0.000} C_DIS
LIN {X 94.390,Y -45.317,Z -49.925,A -90.000,B 90.000,C 0.000} C_DIS
LIN {X 95.092,Y -45.323,Z -49.310,A -90.000,B 90.000,C 0.000} C_DIS
LIN {X 96.070,Y -45.338,Z -48.453,A -90.000,B 90.000,C 0.000} C_DIS
LIN {X 96.236,Y -45.344,Z -48.292,A -90.000,B 90.000,C 0.000} C_DIS
LIN {X 96.855,Y -45.364,Z -47.712,A -90.000,B 90.000,C 0.000} C_DIS
LIN {X 97.344,Y -45.387,Z -47.256,A -90.000,B 90.000,C 0.000} C_DIS
LIN {X 97.651,Y -45.402,Z -46.979,A -90.000,B 90.000,C 0.000} C_DIS
LIN {X 97.914,Y -45.414,Z -46.749,A -90.000,B 90.000,C 0.000} C_DIS
LIN {X 98.218,Y -45.434,Z -46.470,A -90.000,B 90.000,C 0.000} C_DIS
LIN {X 98.431,Y -45.453,Z -46.275,A -90.000,B 90.000,C 0.000} C_DIS
LIN {X 98.957,Y -45.491,Z -45.838,A -90.000,B 90.000,C 0.000} C_DIS
LIN {X 99.147,Y -45.507,Z -45.681,A -90.000,B 90.000,C 0.000} C_DIS
LIN {X 99.495,Y -45.537,Z -45.410,A -90.000,B 90.000,C 0.000} C_DIS
LIN {X 99.962,Y -45.586,Z -45.062,A -90.000,B 90.000,C 0.000} C_DIS
LIN {X 100.053,Y -45.597,Z -44.995,A -90.000,B 90.000,C 0.000} C_DIS
LIN {X 100.392,Y -45.623,Z -44.767,A -90.000,B 90.000,C 0.000} C_DIS
LIN {X 100.659,Y -45.657,Z -44.597,A -90.000,B 90.000,C 0.000} C_DIS
LIN {X 100.873,Y -45.688,Z -44.463,A -90.000,B 90.000,C 0.000} C_DIS
LIN {X 101.059,Y -45.710,Z -44.356,A -90.000,B 90.000,C 0.000} C_DIS
LIN {X 101.291,Y -45.738,Z -44.227,A -90.000,B 90.000,C 0.000} C_DIS
LIN {X 101.614,Y -45.776,Z -44.061,A -90.000,B 90.000,C 0.000} C_DIS
LIN {X 101.945,Y -45.830,Z -43.908,A -90.000,B 90.000,C 0.000} C_DIS
LIN {X 102.183,Y -45.869,Z -43.800,A -90.000,B 90.000,C 0.000} C_DIS
LIN {X 102.333,Y -45.887,Z -43.744,A -90.000,B 90.000,C 0.000} C_DIS
LIN {X 102.668,Y -45.936,Z -43.624,A -90.000,B 90.000,C 0.000} C_DIS
LIN {X 102.734,Y -45.947,Z -43.601,A -90.000,B 90.000,C 0.000} C_DIS
LIN {X 102.826,Y -45.965,Z -43.572,A -90.000,B 90.000,C 0.000} C_DIS
LIN {X 103.150,Y -46.016,Z -43.495,A -90.000,B 90.000,C 0.000} C_DIS
LIN {X 103.348,Y -46.045,Z -43.452,A -90.000,B 90.000,C 0.000} C_DIS
LIN {X 103.706,Y -46.103,Z -43.383,A -90.000,B 90.000,C 0.000} C_DIS
LIN {X 103.807,Y -46.114,Z -43.372,A -90.000,B 90.000,C 0.000} C_DIS
LIN {X 103.947,Y -46.135,Z -43.363,A -90.000,B 90.000,C 0.000} C_DIS
LIN {X 104.191,Y -46.175,Z -43.354,A -90.000,B 90.000,C 0.000} C_DIS
LIN {X 104.351,Y -46.200,Z -43.351,A -90.000,B 90.000,C 0.000} C_DIS
LIN {X 104.488,Y -46.227,Z -43.355,A -90.000,B 90.000,C 0.000} C_DIS
LIN {X 104.871,Y -46.281,Z -43.406,A -90.000,B 90.000,C 0.000} C_DIS
LIN {X 105.087,Y -46.316,Z -43.443,A -90.000,B 90.000,C 0.000} C_DIS
LIN {X 105.167,Y -46.329,Z -43.458,A -90.000,B 90.000,C 0.000} C_DIS
LIN {X 105.216,Y -46.333,Z -43.469,A -90.000,B 90.000,C 0.000} C_DIS
LIN {X 105.370,Y -46.351,Z -43.510,A -90.000,B 90.000,C 0.000} C_DIS
LIN {X 105.465,Y -46.364,Z -43.541,A -90.000,B 90.000,C 0.000} C_DIS
LIN {X 105.779,Y -46.391,Z -43.658,A -90.000,B 90.000,C 0.000} C_DIS
LIN {X 105.896,Y -46.403,Z -43.710,A -90.000,B 90.000,C 0.000} C_DIS
LIN {X 106.004,Y -46.417,Z -43.764,A -90.000,B 90.000,C 0.000} C_DIS
LIN {X 106.191,Y -46.428,Z -43.863,A -90.000,B 90.000,C 0.000} C_DIS
LIN {X 106.465,Y -46.448,Z -44.021,A -90.000,B 90.000,C 0.000} C_DIS
LIN {X 106.605,Y -46.451,Z -44.116,A -90.000,B 90.000,C 0.000} C_DIS
LIN {X 106.720,Y -46.458,Z -44.207,A -90.000,B 90.000,C 0.000} C_DIS
LIN {X 106.962,Y -46.458,Z -44.415,A -90.000,B 90.000,C 0.000} C_DIS
LIN {X 107.082,Y -46.453,Z -44.537,A -90.000,B 90.000,C 0.000} C_DIS
LIN {X 107.179,Y -46.452,Z -44.648,A -90.000,B 90.000,C 0.000} C_DIS
LIN {X 107.372,Y -46.434,Z -44.892,A -90.000,B 90.000,C 0.000} C_DIS
LIN {X 107.447,Y -46.421,Z -45.005,A -90.000,B 90.000,C 0.000} C_DIS
LIN {X 107.530,Y -46.410,Z -45.148,A -90.000,B 90.000,C 0.000} C_DIS
LIN {X 107.598,Y -46.393,Z -45.278,A -90.000,B 90.000,C 0.000} C_DIS
LIN {X 107.671,Y -46.381,Z -45.410,A -90.000,B 90.000,C 0.000} C_DIS
LIN {X 107.724,Y -46.368,Z -45.526,A -90.000,B 90.000,C 0.000} C_DIS
LIN {X 107.796,Y -46.354,Z -45.716,A -90.000,B 90.000,C 0.000} C_DIS
LIN {X 107.880,Y -46.336,Z -45.947,A -90.000,B 90.000,C 0.000} C_DIS
LIN {X 107.897,Y -46.333,Z -45.998,A -90.000,B 90.000,C 0.000} C_DIS
LIN {X 107.980,Y -46.295,Z -46.284,A -90.000,B 90.000,C 0.000} C_DIS
LIN {X 107.991,Y -46.287,Z -46.334,A -90.000,B 90.000,C 0.000} C_DIS
LIN {X 108.012,Y -46.270,Z -46.442,A -90.000,B 90.000,C 0.000} C_DIS
LIN {X 108.081,Y -46.213,Z -46.855,A -90.000,B 90.000,C 0.000} C_DIS
LIN {X 108.115,Y -46.176,Z -47.122,A -90.000,B 90.000,C 0.000} C_DIS
LIN {X 108.137,Y -46.153,Z -47.304,A -90.000,B 90.000,C 0.000} C_DIS
LIN {X 108.139,Y -46.147,Z -47.346,A -90.000,B 90.000,C 0.000} C_DIS
LIN {X 108.142,Y -46.132,Z -47.482,A -90.000,B 90.000,C 0.000} C_DIS
LIN {X 108.140,Y -46.088,Z -47.951,A -90.000,B 90.000,C 0.000} C_DIS
LIN {X 108.130,Y -46.062,Z -48.342,A -90.000,B 90.000,C 0.000} C_DIS
LIN {X 108.124,Y -46.056,Z -48.460,A -90.000,B 90.000,C 0.000} C_DIS
LIN {X 108.117,Y -46.053,Z -48.547,A -90.000,B 90.000,C 0.000} C_DIS
LIN {X 108.116,Y -46.053,Z -48.600,A -90.000,B 90.000,C 0.000} C_DIS
LIN {X 108.123,Y -46.070,Z -48.736,A -90.000,B 90.000,C 0.000} C_DIS
LIN {X 108.138,Y -46.118,Z -49.151,A -90.000,B 90.000,C 0.000} C_DIS
LIN {X 108.149,Y -46.146,Z -49.373,A -90.000,B 90.000,C 0.000} C_DIS
LIN {X 108.149,Y -46.160,Z -49.468,A -90.000,B 90.000,C 0.000} C_DIS
LIN {X 108.134,Y -46.218,Z -49.899,A -90.000,B 90.000,C 0.000} C_DIS
LIN {X 108.114,Y -46.266,Z -50.336,A -90.000,B 90.000,C 0.000} C_DIS
LIN {X 108.105,Y -46.285,Z -50.501,A -90.000,B 90.000,C 0.000} C_DIS
LIN {X 108.089,Y -46.303,Z -50.717,A -90.000,B 90.000,C 0.000} C_DIS
LIN {X 108.062,Y -46.329,Z -51.038,A -90.000,B 90.000,C 0.000} C_DIS
LIN {X 108.039,Y -46.347,Z -51.260,A -90.000,B 90.000,C 0.000} C_DIS
LIN {X 108.004,Y -46.372,Z -51.675,A -90.000,B 90.000,C 0.000} C_DIS
LIN {X 108.003,Y -46.374,Z -51.850,A -90.000,B 90.000,C 0.000} C_DIS
LIN {X 108.002,Y -46.372,Z -51.888,A -90.000,B 90.000,C 0.000} C_DIS
LIN {X 108.004,Y -46.364,Z -52.028,A -90.000,B 90.000,C 0.000} C_DIS
LIN {X 107.995,Y -46.332,Z -52.619,A -90.000,B 90.000,C 0.000} C_DIS
LIN {X 107.994,Y -46.330,Z -52.670,A -90.000,B 90.000,C 0.000} C_DIS
LIN {X 107.994,Y -46.323,Z -52.764,A -90.000,B 90.000,C 0.000} C_DIS
LIN {X 107.988,Y -46.314,Z -52.950,A -90.000,B 90.000,C 0.000} C_DIS
LIN {X 107.971,Y -46.301,Z -53.203,A -90.000,B 90.000,C 0.000} C_DIS
LIN {X 107.938,Y -46.268,Z -53.599,A -90.000,B 90.000,C 0.000} C_DIS
LIN {X 107.916,Y -46.257,Z -53.789,A -90.000,B 90.000,C 0.000} C_DIS
LIN {X 107.910,Y -46.255,Z -53.829,A -90.000,B 90.000,C 0.000} C_DIS
LIN {X 107.831,Y -46.208,Z -54.340,A -90.000,B 90.000,C 0.000} C_DIS
LIN {X 107.804,Y -46.199,Z -54.488,A -90.000,B 90.000,C 0.000} C_DIS
LIN {X 107.670,Y -46.177,Z -55.106,A -90.000,B 90.000,C 0.000} C_DIS
